// mobject-datatypes/Primitive/_LWORD
{attribute 'linkalways'} 
{attribute 'no_explicit_call' := 'This FB is a CLASS and must be accessed using methods or properties'}
{attribute 'enable_dynamic_creation'}
FUNCTION_BLOCK _LWORD EXTENDS NumericDatatypeBase
VAR
	localData : LWORD;
	activeData : REFERENCE TO LWORD REF= localData;
END_VAR

METHOD FB_init : BOOL
VAR_INPUT
	bInitRetains : BOOL; // if TRUE, the retain variables are initialized (warm start / cold start)
	bInCopyCode : BOOL;  // if TRUE, the instance afterwards gets moved WORDo the copy code (online change)
	InitialValue : LWORD;
END_VAR
localData := InitialValue;
END_METHOD

METHOD PROTECTED SerializeMaxValue
VAR_INPUT
	Serializer : I_Serializer;
END_VAR
Serializer.AddLword(MaxValue);
END_METHOD

METHOD PROTECTED SerializeMinValue
VAR_INPUT
	Serializer : I_Serializer;
END_VAR
Serializer.AddLword(MinValue);
END_METHOD

PROPERTY PUBLIC Address : PVOID
GET
Address := ADR(activeData);
END_GET
END_PROPERTY

METHOD PUBLIC ClearReference
VAR_INPUT
END_VAR
activeData REF= localData;
END_METHOD

METHOD PUBLIC Clone : I_Datatype
VAR
    pClone : POINTER TO _LWORD;
END_VAR
pClone := __NEW(_LWORD(InitialValue := Value));
Clone := pClone^;
END_METHOD

PROPERTY PUBLIC IsEven : BOOL
GET
IsEven := (Value mod 2) = 0;
END_GET
END_PROPERTY

PROPERTY PUBLIC IsFloat : BOOL
GET
IsFloat := FALSE;
END_GET
END_PROPERTY

PROPERTY PUBLIC IsSigned : BOOL
GET
IsSigned := FALSE;
END_GET
END_PROPERTY

METHOD PUBLIC MakeReferenceTo
VAR_INPUT
	ReferenceTarget : REFERENCE TO LWORD;
END_VAR
activeData REF= ReferenceTarget;
END_METHOD

PROPERTY PUBLIC MaxValue : LWORD
GET
MaxValue :=  DatatypeLimits.LWORD_MAX_VALUE;
END_GET
END_PROPERTY

PROPERTY PUBLIC MinValue : LWORD
GET
MinValue := DatatypeLimits.LWORD_MIN_VALUE;
END_GET
END_PROPERTY

METHOD PUBLIC SerializeWith
VAR_INPUT
	Serializer : I_Serializer;
END_VAR
Serializer.AddLword(activeData);
END_METHOD

PROPERTY PUBLIC Size : UDINT
GET
Size := SIZEOF(activeData);
END_GET
END_PROPERTY

METHOD TryDeserializeFrom : BOOL
VAR_INPUT
	Deserializer : I_Deserializer;
	Feedback : I_DeserializerFeedback;
END_VAR
TryDeserializeFrom := Deserializer.TryGetLword(activeData, Feedback);
END_METHOD

METHOD TryMakeReferenceTo : BOOL
VAR_INPUT
	Target : I_Datatype;
END_VAR
VAR
	pTargetData : POINTER TO LWORD;
END_VAR
IF NOT IsEquivalentTo(Target) THEN
	RETURN;
END_IF

pTargetData := Target.Address;
activeData REF= pTargetData^;
TryMakeReferenceTo := TRUE;
END_METHOD

PROPERTY PUBLIC TypeName : T_MAXSTRING
GET
TypeName := 'LWORD';
END_GET
END_PROPERTY

PROPERTY PUBLIC Value : REFERENCE TO LWORD
GET
Value REF= activeData;
END_GET
END_PROPERTY

END_FUNCTION_BLOCK

// mobject-converters/Converters/BOOL_TO_/TryConvert_BOOL_TO_SINT
FUNCTION TryConvert_BOOL_TO_SINT : BOOL
VAR_INPUT
	in : BOOL;
	out : REFERENCE TO SINT;
END_VAR

out := BOOL_TO_SINT(in);
TryConvert_BOOL_TO_SINT := TRUE;

END_FUNCTION

// mobject-datatypes/Primitive/_SINT
{attribute 'linkalways'} 
{attribute 'no_explicit_call' := 'This FB is a CLASS and must be accessed using methods or properties'}
{attribute 'enable_dynamic_creation'}
FUNCTION_BLOCK _SINT EXTENDS NumericDatatypeBase
VAR
	localData : SINT;
	activeData : REFERENCE TO SINT REF= localData;
END_VAR

METHOD FB_init : BOOL
VAR_INPUT
	bInitRetains : BOOL; // if TRUE, the retain variables are initialized (warm start / cold start)
	bInCopyCode : BOOL;  // if TRUE, the instance afterwards gets moved into the copy code (online change)
	InitialValue : SINT;
END_VAR
localData := InitialValue;
END_METHOD

METHOD PROTECTED SerializeMaxValue
VAR_INPUT
	Serializer : I_Serializer;
END_VAR
Serializer.AddSint(MaxValue);
END_METHOD

METHOD PROTECTED SerializeMinValue
VAR_INPUT
	Serializer : I_Serializer;
END_VAR
Serializer.AddSint(MinValue);
END_METHOD

PROPERTY PUBLIC Address : PVOID
GET
Address := ADR(activeData);
END_GET
END_PROPERTY

METHOD PUBLIC ClearReference
VAR_INPUT
END_VAR
activeData REF= localData;
END_METHOD

METHOD PUBLIC Clone : I_Datatype
VAR
    pClone : POINTER TO _SINT;
END_VAR
pClone := __NEW(_SINT(InitialValue := Value));
Clone := pClone^;
END_METHOD

PROPERTY PUBLIC IsEven : BOOL
GET
IsEven := (Value mod 2) = 0;
END_GET
END_PROPERTY

PROPERTY PUBLIC IsFloat : BOOL
GET
IsFloat := FALSE;
END_GET
END_PROPERTY

PROPERTY PUBLIC IsSigned : BOOL
GET
IsSigned := TRUE;
END_GET
END_PROPERTY

METHOD PUBLIC MakeReferenceTo
VAR_INPUT
	ReferenceTarget : REFERENCE TO SINT;
END_VAR
activeData REF= ReferenceTarget;
END_METHOD

PROPERTY PUBLIC MaxValue : SINT
GET
MaxValue :=  DatatypeLimits.SINT_MAX_VALUE;
END_GET
END_PROPERTY

PROPERTY PUBLIC MinValue : SINT
GET
MinValue := DatatypeLimits.SINT_MIN_VALUE;
END_GET
END_PROPERTY

METHOD PUBLIC SerializeWith
VAR_INPUT
	Serializer : I_Serializer;
END_VAR
Serializer.AddSint(activeData);
END_METHOD

PROPERTY PUBLIC Size : UDINT
GET
Size := SIZEOF(activeData);
END_GET
END_PROPERTY

METHOD TryDeserializeFrom : BOOL
VAR_INPUT
	Deserializer : I_Deserializer;
	Feedback : I_DeserializerFeedback;
END_VAR
TryDeserializeFrom := Deserializer.TryGetSint(activeData, Feedback);
END_METHOD

METHOD TryMakeReferenceTo : BOOL
VAR_INPUT
	Target : I_Datatype;
END_VAR
VAR
	pTargetData : POINTER TO SINT;
END_VAR
IF NOT IsEquivalentTo(Target) THEN
	RETURN;
END_IF

pTargetData := Target.Address;
activeData REF= pTargetData^;
TryMakeReferenceTo := TRUE;
END_METHOD

PROPERTY PUBLIC TypeName : T_MAXSTRING
GET
TypeName := 'SINT';
END_GET
END_PROPERTY

PROPERTY PUBLIC Value : REFERENCE TO SINT
GET
Value REF= activeData;
END_GET
END_PROPERTY

END_FUNCTION_BLOCK

// mobject-converters/Converters/BOOL_TO_/TryConvert_BOOL_TO_INT
FUNCTION TryConvert_BOOL_TO_INT : BOOL
VAR_INPUT
	in : BOOL;
	out : REFERENCE TO INT;
END_VAR

out := BOOL_TO_INT(in);
TryConvert_BOOL_TO_INT := TRUE;

END_FUNCTION

// mobject-datatypes/Primitive/_INT
{attribute 'linkalways'} 
{attribute 'no_explicit_call' := 'This FB is a CLASS and must be accessed using methods or properties'}
{attribute 'enable_dynamic_creation'}
FUNCTION_BLOCK _INT EXTENDS NumericDatatypeBase
VAR
	localData : INT;
	activeData : REFERENCE TO INT REF= localData;
END_VAR

METHOD FB_init : BOOL
VAR_INPUT
	bInitRetains : BOOL; // if TRUE, the retain variables are initialized (warm start / cold start)
	bInCopyCode : BOOL;  // if TRUE, the instance afterwards gets moved into the copy code (online change)
	InitialValue : INT;
END_VAR
localData := InitialValue;
END_METHOD

METHOD PROTECTED SerializeMaxValue
VAR_INPUT
	Serializer : I_Serializer;
END_VAR
Serializer.AddInt(MaxValue);
END_METHOD

METHOD PROTECTED SerializeMinValue
VAR_INPUT
	Serializer : I_Serializer;
END_VAR
Serializer.AddInt(MinValue);
END_METHOD

PROPERTY PUBLIC Address : PVOID
GET
Address := ADR(activeData);
END_GET
END_PROPERTY

METHOD PUBLIC ClearReference
VAR_INPUT
END_VAR
activeData REF= localData;
END_METHOD

METHOD PUBLIC Clone : I_Datatype
VAR
    pClone : POINTER TO _INT;
END_VAR
pClone := __NEW(_INT(InitialValue := Value));
Clone := pClone^;
END_METHOD

PROPERTY PUBLIC IsEven : BOOL
GET
IsEven := (Value mod 2) = 0;
END_GET
END_PROPERTY

PROPERTY PUBLIC IsFloat : BOOL
GET
IsFloat := FALSE;
END_GET
END_PROPERTY

PROPERTY PUBLIC IsSigned : BOOL
GET
IsSigned := TRUE;
END_GET
END_PROPERTY

METHOD PUBLIC MakeReferenceTo
VAR_INPUT
	ReferenceTarget : REFERENCE TO INT;
END_VAR
activeData REF= ReferenceTarget;
END_METHOD

PROPERTY PUBLIC MaxValue : INT
GET
MaxValue := DatatypeLimits.INT_MAX_VALUE;
END_GET
END_PROPERTY

PROPERTY PUBLIC MinValue : INT
GET
MinValue := DatatypeLimits.INT_MIN_VALUE;
END_GET
END_PROPERTY

METHOD PUBLIC SerializeWith
VAR_INPUT
	Serializer : I_Serializer;
END_VAR
Serializer.AddInt(activeData);
END_METHOD

PROPERTY PUBLIC Size : UDINT
GET
Size := SIZEOF(activeData);
END_GET
END_PROPERTY

METHOD TryDeserializeFrom : BOOL
VAR_INPUT
	Deserializer : I_Deserializer;
	Feedback : I_DeserializerFeedback;
END_VAR
TryDeserializeFrom := Deserializer.TryGetInt(activeData, Feedback);
END_METHOD

METHOD TryMakeReferenceTo : BOOL
VAR_INPUT
	Target : I_Datatype;
END_VAR
VAR
	pTargetData : POINTER TO INT;
END_VAR
IF NOT IsEquivalentTo(Target) THEN
	RETURN;
END_IF

pTargetData := Target.Address;
activeData REF= pTargetData^;
TryMakeReferenceTo := TRUE;
END_METHOD

PROPERTY PUBLIC TypeName : T_MAXSTRING
GET
TypeName := 'INT';
END_GET
END_PROPERTY

PROPERTY PUBLIC Value : REFERENCE TO INT
GET
Value REF= activeData;
END_GET
END_PROPERTY

END_FUNCTION_BLOCK

// mobject-converters/Converters/BOOL_TO_/TryConvert_BOOL_TO_DINT
FUNCTION TryConvert_BOOL_TO_DINT : BOOL
VAR_INPUT
	in : BOOL;
	out : REFERENCE TO DINT;
END_VAR

out := BOOL_TO_DINT(in);
TryConvert_BOOL_TO_DINT := TRUE;

END_FUNCTION

// mobject-datatypes/Primitive/_DINT
{attribute 'linkalways'} 
{attribute 'no_explicit_call' := 'This FB is a CLASS and must be accessed using methods or properties'}
{attribute 'enable_dynamic_creation'}
FUNCTION_BLOCK _DINT EXTENDS NumericDatatypeBase
VAR
	localData : DINT;
	activeData : REFERENCE TO DINT REF= localData;
END_VAR

METHOD FB_init : BOOL
VAR_INPUT
	bInitRetains : BOOL; // if TRUE, the retain variables are initialized (warm start / cold start)
	bInCopyCode : BOOL;  // if TRUE, the instance afterwards gets moved into the copy code (online change)
	InitialValue : DINT;
END_VAR
localData := InitialValue;
END_METHOD

METHOD PROTECTED SerializeMaxValue
VAR_INPUT
	Serializer : I_Serializer;
END_VAR
Serializer.AddDint(MaxValue);
END_METHOD

METHOD PROTECTED SerializeMinValue
VAR_INPUT
	Serializer : I_Serializer;
END_VAR
Serializer.AddDint(MinValue);
END_METHOD

PROPERTY PUBLIC Address : PVOID
GET
Address := ADR(activeData);
END_GET
END_PROPERTY

METHOD PUBLIC ClearReference
VAR_INPUT
END_VAR
activeData REF= localData;
END_METHOD

METHOD PUBLIC Clone : I_Datatype
VAR
    pClone : POINTER TO _DINT;
END_VAR
pClone := __NEW(_DINT(InitialValue := Value));
Clone := pClone^;
END_METHOD

PROPERTY PUBLIC IsEven : BOOL
GET
IsEven := (Value mod 2) = 0;
END_GET
END_PROPERTY

PROPERTY PUBLIC IsFloat : BOOL
GET
IsFloat := FALSE;
END_GET
END_PROPERTY

PROPERTY PUBLIC IsSigned : BOOL
GET
IsSigned := TRUE;
END_GET
END_PROPERTY

METHOD PUBLIC MakeReferenceTo
VAR_INPUT
	ReferenceTarget : REFERENCE TO DINT;
END_VAR
activeData REF= ReferenceTarget;
END_METHOD

PROPERTY PUBLIC MaxValue : DINT
GET
MaxValue := DatatypeLimits.DINT_MAX_VALUE;
END_GET
END_PROPERTY

PROPERTY PUBLIC MinValue : DINT
GET
MinValue := DatatypeLimits.DINT_MIN_VALUE;
END_GET
END_PROPERTY

METHOD PUBLIC SerializeWith
VAR_INPUT
	Serializer : I_Serializer;
END_VAR
Serializer.AddDint(activeData);
END_METHOD

PROPERTY PUBLIC Size : UDINT
GET
Size := SIZEOF(activeData);
END_GET
END_PROPERTY

METHOD TryDeserializeFrom : BOOL
VAR_INPUT
	Deserializer : I_Deserializer;
	Feedback : I_DeserializerFeedback;
END_VAR
TryDeserializeFrom := Deserializer.TryGetDint(activeData, Feedback);
END_METHOD

METHOD TryMakeReferenceTo : BOOL
VAR_INPUT
	Target : I_Datatype;
END_VAR
VAR
	pTargetData : POINTER TO DINT;
END_VAR
IF NOT IsEquivalentTo(Target) THEN
	RETURN;
END_IF

pTargetData := Target.Address;
activeData REF= pTargetData^;
TryMakeReferenceTo := TRUE;
END_METHOD

PROPERTY PUBLIC TypeName : T_MAXSTRING
GET
TypeName := 'DINT';
END_GET
END_PROPERTY

PROPERTY PUBLIC Value : REFERENCE TO DINT
GET
Value REF= activeData;
END_GET
END_PROPERTY

END_FUNCTION_BLOCK

// mobject-converters/Converters/BOOL_TO_/TryConvert_BOOL_TO_LINT
FUNCTION TryConvert_BOOL_TO_LINT : BOOL
VAR_INPUT
	in : BOOL;
	out : REFERENCE TO LINT;
END_VAR

out := BOOL_TO_LINT(in);
TryConvert_BOOL_TO_LINT := TRUE;

END_FUNCTION

// mobject-datatypes/Primitive/_LINT
{attribute 'linkalways'} 
{attribute 'no_explicit_call' := 'This FB is a CLASS and must be accessed using methods or properties'}
{attribute 'enable_dynamic_creation'}
FUNCTION_BLOCK _LINT EXTENDS NumericDatatypeBase
VAR
	localData : LINT;
	activeData : REFERENCE TO LINT REF= localData;
END_VAR

METHOD FB_init : BOOL
VAR_INPUT
	bInitRetains : BOOL; // if TRUE, the retain variables are initialized (warm start / cold start)
	bInCopyCode : BOOL;  // if TRUE, the instance afterwards gets moved into the copy code (online change)
	InitialValue : LINT;
END_VAR
localData := InitialValue;
END_METHOD

METHOD PROTECTED SerializeMaxValue
VAR_INPUT
	Serializer : I_Serializer;
END_VAR
Serializer.AddLint(MaxValue);
END_METHOD

METHOD PROTECTED SerializeMinValue
VAR_INPUT
	Serializer : I_Serializer;
END_VAR
Serializer.AddLint(MinValue);
END_METHOD

PROPERTY PUBLIC Address : PVOID
GET
Address := ADR(activeData);
END_GET
END_PROPERTY

METHOD PUBLIC ClearReference
VAR_INPUT
END_VAR
activeData REF= localData;
END_METHOD

METHOD PUBLIC Clone : I_Datatype
VAR
    pClone : POINTER TO _LINT;
END_VAR
pClone := __NEW(_LINT(InitialValue := Value));
Clone := pClone^;
END_METHOD

PROPERTY PUBLIC IsEven : BOOL
GET
IsEven := (Value mod 2) = 0;
END_GET
END_PROPERTY

PROPERTY PUBLIC IsFloat : BOOL
GET
IsFloat := FALSE;
END_GET
END_PROPERTY

PROPERTY PUBLIC IsSigned : BOOL
GET
IsSigned := TRUE;
END_GET
END_PROPERTY

METHOD PUBLIC MakeReferenceTo
VAR_INPUT
	ReferenceTarget : REFERENCE TO LINT;
END_VAR
activeData REF= ReferenceTarget;
END_METHOD

PROPERTY PUBLIC MaxValue : LINT
GET
MaxValue :=  DatatypeLimits.LINT_MAX_VALUE;
END_GET
END_PROPERTY

PROPERTY PUBLIC MinValue : LINT
GET
MinValue := DatatypeLimits.LINT_MIN_VALUE;
END_GET
END_PROPERTY

METHOD PUBLIC SerializeWith
VAR_INPUT
	Serializer : I_Serializer;
END_VAR
Serializer.AddLint(activeData);
END_METHOD

PROPERTY PUBLIC Size : UDINT
GET
Size := SIZEOF(activeData);
END_GET
END_PROPERTY

METHOD TryDeserializeFrom : BOOL
VAR_INPUT
	Deserializer : I_Deserializer;
	Feedback : I_DeserializerFeedback;
END_VAR
TryDeserializeFrom := Deserializer.TryGetLint(activeData, Feedback);
END_METHOD

METHOD TryMakeReferenceTo : BOOL
VAR_INPUT
	Target : I_Datatype;
END_VAR
VAR
	pTargetData : POINTER TO LINT;
END_VAR
IF NOT IsEquivalentTo(Target) THEN
	RETURN;
END_IF

pTargetData := Target.Address;
activeData REF= pTargetData^;
TryMakeReferenceTo := TRUE;
END_METHOD

PROPERTY PUBLIC TypeName : T_MAXSTRING
GET
TypeName := 'LINT';
END_GET
END_PROPERTY

PROPERTY PUBLIC Value : REFERENCE TO LINT
GET
Value REF= activeData;
END_GET
END_PROPERTY

END_FUNCTION_BLOCK

// mobject-converters/Converters/BOOL_TO_/TryConvert_BOOL_TO_USINT
FUNCTION TryConvert_BOOL_TO_USINT : BOOL
VAR_INPUT
	in : BOOL;
	out : REFERENCE TO USINT;
END_VAR

out := BOOL_TO_USINT(in);
TryConvert_BOOL_TO_USINT := TRUE;

END_FUNCTION

// mobject-datatypes/Primitive/_USINT
{attribute 'linkalways'} 
{attribute 'no_explicit_call' := 'This FB is a CLASS and must be accessed using methods or properties'}
{attribute 'enable_dynamic_creation'}
FUNCTION_BLOCK _USINT EXTENDS NumericDatatypeBase
VAR
	localData : USINT;
	activeData : REFERENCE TO USINT REF= localData;
END_VAR

METHOD FB_init : BOOL
VAR_INPUT
	bInitRetains : BOOL; // if TRUE, the retain variables are initialized (warm start / cold start)
	bInCopyCode : BOOL;  // if TRUE, the instance afterwards gets moved into the copy code (online change)
	InitialValue : USINT;
END_VAR
localData := InitialValue;
END_METHOD

METHOD PROTECTED SerializeMaxValue
VAR_INPUT
	Serializer : I_Serializer;
END_VAR
Serializer.AddUsint(MaxValue);
END_METHOD

METHOD PROTECTED SerializeMinValue
VAR_INPUT
	Serializer : I_Serializer;
END_VAR
Serializer.AddUsint(MinValue);
END_METHOD

PROPERTY PUBLIC Address : PVOID
GET
Address := ADR(activeData);
END_GET
END_PROPERTY

METHOD PUBLIC ClearReference
VAR_INPUT
END_VAR
activeData REF= localData;
END_METHOD

METHOD PUBLIC Clone : I_Datatype
VAR
    pClone : POINTER TO _USINT;
END_VAR
pClone := __NEW(_USINT(InitialValue := Value));
Clone := pClone^;
END_METHOD

PROPERTY PUBLIC IsEven : BOOL
GET
IsEven := (Value mod 2) = 0;
END_GET
END_PROPERTY

PROPERTY PUBLIC IsFloat : BOOL
GET
IsFloat := FALSE;
END_GET
END_PROPERTY

PROPERTY PUBLIC IsSigned : BOOL
GET
IsSigned := FALSE;
END_GET
END_PROPERTY

METHOD PUBLIC MakeReferenceTo
VAR_INPUT
	ReferenceTarget : REFERENCE TO USINT;
END_VAR
activeData REF= ReferenceTarget;
END_METHOD

PROPERTY PUBLIC MaxValue : USINT
GET
MaxValue :=  DatatypeLimits.USINT_MAX_VALUE;
END_GET
END_PROPERTY

PROPERTY PUBLIC MinValue : USINT
GET
MinValue := DatatypeLimits.USINT_MIN_VALUE;
END_GET
END_PROPERTY

METHOD PUBLIC SerializeWith
VAR_INPUT
	Serializer : I_Serializer;
END_VAR
Serializer.AddUsint(activeData);
END_METHOD

PROPERTY PUBLIC Size : UDINT
GET
Size := SIZEOF(activeData);
END_GET
END_PROPERTY

METHOD TryDeserializeFrom : BOOL
VAR_INPUT
	Deserializer : I_Deserializer;
	Feedback : I_DeserializerFeedback;
END_VAR
TryDeserializeFrom := Deserializer.TryGetUsint(activeData, Feedback);
END_METHOD

METHOD TryMakeReferenceTo : BOOL
VAR_INPUT
	Target : I_Datatype;
END_VAR
VAR
	pTargetData : POINTER TO USINT;
END_VAR
IF NOT IsEquivalentTo(Target) THEN
	RETURN;
END_IF

pTargetData := Target.Address;
activeData REF= pTargetData^;
TryMakeReferenceTo := TRUE;
END_METHOD

PROPERTY PUBLIC TypeName : T_MAXSTRING
GET
TypeName := 'USINT';
END_GET
END_PROPERTY

PROPERTY PUBLIC Value : REFERENCE TO USINT
GET
Value REF= activeData;
END_GET
END_PROPERTY

END_FUNCTION_BLOCK

// mobject-converters/Converters/BOOL_TO_/TryConvert_BOOL_TO_UINT
FUNCTION TryConvert_BOOL_TO_UINT : BOOL
VAR_INPUT
	in : BOOL;
	out : REFERENCE TO UINT;
END_VAR

out := BOOL_TO_UINT(in);
TryConvert_BOOL_TO_UINT := TRUE;

END_FUNCTION

// mobject-datatypes/Primitive/_UINT
{attribute 'linkalways'} 
{attribute 'no_explicit_call' := 'This FB is a CLASS and must be accessed using methods or properties'}
{attribute 'enable_dynamic_creation'}
FUNCTION_BLOCK _UINT EXTENDS NumericDatatypeBase
VAR
	localData : UINT;
	activeData : REFERENCE TO UINT REF= localData;
END_VAR

METHOD FB_init : BOOL
VAR_INPUT
	bInitRetains : BOOL; // if TRUE, the retain variables are initialized (warm start / cold start)
	bInCopyCode : BOOL;  // if TRUE, the instance afterwards gets moved into the copy code (online change)
	InitialValue : UINT;
END_VAR
localData := InitialValue;
END_METHOD

METHOD PROTECTED SerializeMaxValue
VAR_INPUT
	Serializer : I_Serializer;
END_VAR
Serializer.AddUint(MaxValue);
END_METHOD

METHOD PROTECTED SerializeMinValue
VAR_INPUT
	Serializer : I_Serializer;
END_VAR
Serializer.AddUint(MinValue);
END_METHOD

PROPERTY PUBLIC Address : PVOID
GET
Address := ADR(activeData);
END_GET
END_PROPERTY

METHOD PUBLIC ClearReference
VAR_INPUT
END_VAR
activeData REF= localData;
END_METHOD

METHOD PUBLIC Clone : I_Datatype
VAR
    pClone : POINTER TO _UINT;
END_VAR
pClone := __NEW(_UINT(InitialValue := Value));
Clone := pClone^;
END_METHOD

PROPERTY PUBLIC IsEven : BOOL
GET
IsEven := (Value mod 2) = 0;
END_GET
END_PROPERTY

PROPERTY PUBLIC IsFloat : BOOL
GET
IsFloat := FALSE;
END_GET
END_PROPERTY

PROPERTY PUBLIC IsSigned : BOOL
GET
IsSigned := FALSE;
END_GET
END_PROPERTY

METHOD PUBLIC MakeReferenceTo
VAR_INPUT
	ReferenceTarget : REFERENCE TO UINT;
END_VAR
activeData REF= ReferenceTarget;
END_METHOD

PROPERTY PUBLIC MaxValue : UINT
GET
MaxValue :=  DatatypeLimits.UINT_MAX_VALUE;
END_GET
END_PROPERTY

PROPERTY PUBLIC MinValue : UINT
GET
MinValue := DatatypeLimits.UINT_MIN_VALUE;
END_GET
END_PROPERTY

METHOD PUBLIC SerializeWith
VAR_INPUT
	Serializer : I_Serializer;
END_VAR
Serializer.AddUint(activeData);
END_METHOD

PROPERTY PUBLIC Size : UDINT
GET
Size := SIZEOF(activeData);
END_GET
END_PROPERTY

METHOD TryDeserializeFrom : BOOL
VAR_INPUT
	Deserializer : I_Deserializer;
	Feedback : I_DeserializerFeedback;
END_VAR
TryDeserializeFrom := Deserializer.TryGetUint(activeData, Feedback);
END_METHOD

METHOD TryMakeReferenceTo : BOOL
VAR_INPUT
	Target : I_Datatype;
END_VAR
VAR
	pTargetData : POINTER TO UINT;
END_VAR
IF NOT IsEquivalentTo(Target) THEN
	RETURN;
END_IF

pTargetData := Target.Address;
activeData REF= pTargetData^;
TryMakeReferenceTo := TRUE;
END_METHOD

PROPERTY PUBLIC TypeName : T_MAXSTRING
GET
TypeName := 'UINT';
END_GET
END_PROPERTY

PROPERTY PUBLIC Value : REFERENCE TO UINT
GET
Value REF= activeData;
END_GET
END_PROPERTY

END_FUNCTION_BLOCK

// mobject-converters/Converters/BOOL_TO_/TryConvert_BOOL_TO_UDINT
FUNCTION TryConvert_BOOL_TO_UDINT : BOOL
VAR_INPUT
	in : BOOL;
	out : REFERENCE TO UDINT;
END_VAR

out := BOOL_TO_UDINT(in);
TryConvert_BOOL_TO_UDINT := TRUE;

END_FUNCTION

// mobject-datatypes/Primitive/_UDINT
{attribute 'linkalways'} 
{attribute 'no_explicit_call' := 'This FB is a CLASS and must be accessed using methods or properties'}
{attribute 'enable_dynamic_creation'}
FUNCTION_BLOCK _UDINT EXTENDS NumericDatatypeBase
VAR
	localData : UDINT;
	activeData : REFERENCE TO UDINT REF= localData;
END_VAR

METHOD FB_init : BOOL
VAR_INPUT
	bInitRetains : BOOL; // if TRUE, the retain variables are initialized (warm start / cold start)
	bInCopyCode : BOOL;  // if TRUE, the instance afterwards gets moved into the copy code (online change)
	InitialValue : UDINT;
END_VAR
localData := InitialValue;
END_METHOD

METHOD PROTECTED SerializeMaxValue
VAR_INPUT
	Serializer : I_Serializer;
END_VAR
Serializer.AddUdint(MaxValue);
END_METHOD

METHOD PROTECTED SerializeMinValue
VAR_INPUT
	Serializer : I_Serializer;
END_VAR
Serializer.AddUdint(MinValue);
END_METHOD

PROPERTY PUBLIC Address : PVOID
GET
Address := ADR(activeData);
END_GET
END_PROPERTY

METHOD PUBLIC ClearReference
VAR_INPUT
END_VAR
activeData REF= localData;
END_METHOD

METHOD PUBLIC Clone : I_Datatype
VAR
    pClone : POINTER TO _UDINT;
END_VAR
pClone := __NEW(_UDINT(InitialValue := Value));
Clone := pClone^;
END_METHOD

PROPERTY PUBLIC IsEven : BOOL
GET
IsEven := (Value mod 2) = 0;
END_GET
END_PROPERTY

PROPERTY PUBLIC IsFloat : BOOL
GET
IsFloat := FALSE;
END_GET
END_PROPERTY

PROPERTY PUBLIC IsSigned : BOOL
GET
IsSigned := FALSE;
END_GET
END_PROPERTY

METHOD PUBLIC MakeReferenceTo
VAR_INPUT
	ReferenceTarget : REFERENCE TO UDINT;
END_VAR
activeData REF= ReferenceTarget;
END_METHOD

PROPERTY PUBLIC MaxValue : UDINT
GET
MaxValue :=  DatatypeLimits.UDINT_MAX_VALUE;
END_GET
END_PROPERTY

PROPERTY PUBLIC MinValue : UDINT
GET
MinValue := DatatypeLimits.UDINT_MIN_VALUE;
END_GET
END_PROPERTY

METHOD PUBLIC SerializeWith
VAR_INPUT
	Serializer : I_Serializer;
END_VAR
Serializer.AddUdint(activeData);
END_METHOD

PROPERTY PUBLIC Size : UDINT
GET
Size := SIZEOF(activeData);
END_GET
END_PROPERTY

METHOD TryDeserializeFrom : BOOL
VAR_INPUT
	Deserializer : I_Deserializer;
	Feedback : I_DeserializerFeedback;
END_VAR
TryDeserializeFrom := Deserializer.TryGetUdint(activeData, Feedback);
END_METHOD

METHOD TryMakeReferenceTo : BOOL
VAR_INPUT
	Target : I_Datatype;
END_VAR
VAR
	pTargetData : POINTER TO UDINT;
END_VAR
IF NOT IsEquivalentTo(Target) THEN
	RETURN;
END_IF

pTargetData := Target.Address;
activeData REF= pTargetData^;
TryMakeReferenceTo := TRUE;
END_METHOD

PROPERTY PUBLIC TypeName : T_MAXSTRING
GET
TypeName := 'UDINT';
END_GET
END_PROPERTY

PROPERTY PUBLIC Value : REFERENCE TO UDINT
GET
Value REF= activeData;
END_GET
END_PROPERTY

END_FUNCTION_BLOCK

// mobject-converters/Converters/BOOL_TO_/TryConvert_BOOL_TO_ULINT
FUNCTION TryConvert_BOOL_TO_ULINT : BOOL
VAR_INPUT
	in : BOOL;
	out : REFERENCE TO ULINT;
END_VAR

out := BOOL_TO_ULINT(in);
TryConvert_BOOL_TO_ULINT := TRUE;

END_FUNCTION

// mobject-datatypes/Primitive/_ULINT
{attribute 'linkalways'} 
{attribute 'no_explicit_call' := 'This FB is a CLASS and must be accessed using methods or properties'}
{attribute 'enable_dynamic_creation'}
FUNCTION_BLOCK _ULINT EXTENDS NumericDatatypeBase
VAR
	localData : ULINT;
	activeData : REFERENCE TO ULINT REF= localData;
END_VAR

METHOD FB_init : BOOL
VAR_INPUT
	bInitRetains : BOOL; // if TRUE, the retain variables are initialized (warm start / cold start)
	bInCopyCode : BOOL;  // if TRUE, the instance afterwards gets moved into the copy code (online change)
	InitialValue : ULINT;
END_VAR
localData := InitialValue;
END_METHOD

METHOD PROTECTED SerializeMaxValue
VAR_INPUT
	Serializer : I_Serializer;
END_VAR
Serializer.AddUlint(MaxValue);
END_METHOD

METHOD PROTECTED SerializeMinValue
VAR_INPUT
	Serializer : I_Serializer;
END_VAR
Serializer.AddUlint(MinValue);
END_METHOD

PROPERTY PUBLIC Address : PVOID
GET
Address := ADR(activeData);
END_GET
END_PROPERTY

METHOD PUBLIC ClearReference
VAR_INPUT
END_VAR
activeData REF= localData;
END_METHOD

METHOD PUBLIC Clone : I_Datatype
VAR
    pClone : POINTER TO _ULINT;
END_VAR
pClone := __NEW(_ULINT(InitialValue := Value));
Clone := pClone^;
END_METHOD

PROPERTY PUBLIC IsEven : BOOL
GET
IsEven := (Value mod 2) = 0;
END_GET
END_PROPERTY

PROPERTY PUBLIC IsFloat : BOOL
GET
IsFloat := FALSE;
END_GET
END_PROPERTY

PROPERTY PUBLIC IsSigned : BOOL
GET
IsSigned := FALSE;
END_GET
END_PROPERTY

METHOD PUBLIC MakeReferenceTo
VAR_INPUT
	ReferenceTarget : REFERENCE TO ULINT;
END_VAR
activeData REF= ReferenceTarget;
END_METHOD

PROPERTY PUBLIC MaxValue : ULINT
GET
MaxValue :=  DatatypeLimits.ULINT_MAX_VALUE;
END_GET
END_PROPERTY

PROPERTY PUBLIC MinValue : ULINT
GET
MinValue := DatatypeLimits.ULINT_MIN_VALUE;
END_GET
END_PROPERTY

METHOD PUBLIC SerializeWith
VAR_INPUT
	Serializer : I_Serializer;
END_VAR
Serializer.AddUlint(activeData);
END_METHOD

PROPERTY PUBLIC Size : UDINT
GET
Size := SIZEOF(activeData);
END_GET
END_PROPERTY

METHOD TryDeserializeFrom : BOOL
VAR_INPUT
	Deserializer : I_Deserializer;
	Feedback : I_DeserializerFeedback;
END_VAR
TryDeserializeFrom := Deserializer.TryGetUlint(activeData, Feedback);
END_METHOD

METHOD TryMakeReferenceTo : BOOL
VAR_INPUT
	Target : I_Datatype;
END_VAR
VAR
	pTargetData : POINTER TO ULINT;
END_VAR
IF NOT IsEquivalentTo(Target) THEN
	RETURN;
END_IF

pTargetData := Target.Address;
activeData REF= pTargetData^;
TryMakeReferenceTo := TRUE;
END_METHOD

PROPERTY PUBLIC TypeName : T_MAXSTRING
GET
TypeName := 'ULINT';
END_GET
END_PROPERTY

PROPERTY PUBLIC Value : REFERENCE TO ULINT
GET
Value REF= activeData;
END_GET
END_PROPERTY

END_FUNCTION_BLOCK

// mobject-converters/Converters/BOOL_TO_/TryConvert_BOOL_TO_REAL
FUNCTION TryConvert_BOOL_TO_REAL : BOOL
VAR_INPUT
	in : BOOL;
	out : REFERENCE TO REAL;
END_VAR

out := BOOL_TO_REAL(in);
TryConvert_BOOL_TO_REAL := TRUE;

END_FUNCTION

// mobject-datatypes/Primitive/_REAL
{attribute 'linkalways'} 
{attribute 'no_explicit_call' := 'This FB is a CLASS and must be accessed using methods or properties'}
{attribute 'enable_dynamic_creation'}
FUNCTION_BLOCK _REAL EXTENDS NumericDatatypeBase
VAR
	localData : REAL;
	activeData : REFERENCE TO REAL REF= localData;
END_VAR

METHOD FB_init : BOOL
VAR_INPUT
	bInitRetains : BOOL; // if TRUE, the retain variables are initialized (warm start / cold start)
	bInCopyCode : BOOL;  // if TRUE, the instance afterwards gets moved into the copy code (online change)
	InitialValue : REAL;
END_VAR
localData := InitialValue;
END_METHOD

METHOD PROTECTED SerializeMaxValue
VAR_INPUT
	Serializer : I_Serializer;
END_VAR
Serializer.AddReal(MaxValue);
END_METHOD

METHOD PROTECTED SerializeMinValue
VAR_INPUT
	Serializer : I_Serializer;
END_VAR
Serializer.AddReal(MinValue);
END_METHOD

PROPERTY PUBLIC Address : PVOID
GET
Address := ADR(activeData);
END_GET
END_PROPERTY

METHOD PUBLIC ClearReference
VAR_INPUT
END_VAR
activeData REF= localData;
END_METHOD

METHOD PUBLIC Clone : I_Datatype
VAR
    pClone : POINTER TO _REAL;
END_VAR
pClone := __NEW(_REAL(InitialValue := Value));
Clone := pClone^;
END_METHOD

PROPERTY PUBLIC IsEven : BOOL
GET
IsEven := FALSE;
END_GET
END_PROPERTY

PROPERTY PUBLIC IsFloat : BOOL
GET
IsFloat := TRUE;
END_GET
END_PROPERTY

PROPERTY PUBLIC IsOdd : BOOL
GET
IsOdd := FALSE;
END_GET
END_PROPERTY

PROPERTY PUBLIC IsSigned : BOOL
GET
IsSigned := TRUE;
END_GET
END_PROPERTY

METHOD PUBLIC MakeReferenceTo
VAR_INPUT
	ReferenceTarget : REFERENCE TO REAL;
END_VAR
activeData REF= ReferenceTarget;
END_METHOD

PROPERTY PUBLIC MaxValue : REAL
GET
MaxValue :=  DatatypeLimits.REAL_MAX_VALUE;
END_GET
END_PROPERTY

PROPERTY PUBLIC MinValue : REAL
GET
MinValue := DatatypeLimits.REAL_MIN_VALUE;
END_GET
END_PROPERTY

METHOD PUBLIC SerializeWith
VAR_INPUT
	Serializer : I_Serializer;
END_VAR
Serializer.AddReal(activeData);
END_METHOD

PROPERTY PUBLIC Size : UDINT
GET
Size := SIZEOF(activeData);
END_GET
END_PROPERTY

METHOD TryDeserializeFrom : BOOL
VAR_INPUT
	Deserializer : I_Deserializer;
	Feedback : I_DeserializerFeedback;
END_VAR
TryDeserializeFrom := Deserializer.TryGetReal(activeData, Feedback);
END_METHOD

METHOD TryMakeReferenceTo : BOOL
VAR_INPUT
	Target : I_Datatype;
END_VAR
VAR
	pTargetData : POINTER TO REAL;
END_VAR
IF NOT IsEquivalentTo(Target) THEN
	RETURN;
END_IF

pTargetData := Target.Address;
activeData REF= pTargetData^;
TryMakeReferenceTo := TRUE;
END_METHOD

PROPERTY PUBLIC TypeName : T_MAXSTRING
GET
TypeName := 'REAL';
END_GET
END_PROPERTY

PROPERTY PUBLIC Value : REFERENCE TO REAL
GET
Value REF= activeData;
END_GET
END_PROPERTY

END_FUNCTION_BLOCK

// mobject-converters/Converters/BOOL_TO_/TryConvert_BOOL_TO_LREAL
FUNCTION TryConvert_BOOL_TO_LREAL : BOOL
VAR_INPUT
	in : BOOL;
	out : REFERENCE TO LREAL;
END_VAR

out := BOOL_TO_LREAL(in);
TryConvert_BOOL_TO_LREAL := TRUE;

END_FUNCTION

// mobject-datatypes/Primitive/_LREAL
{attribute 'linkalways'} 
{attribute 'no_explicit_call' := 'This FB is a CLASS and must be accessed using methods or properties'}
{attribute 'enable_dynamic_creation'}
FUNCTION_BLOCK _LREAL EXTENDS NumericDatatypeBase
VAR
	localData : LREAL;
	activeData : REFERENCE TO LREAL REF= localData;
END_VAR

METHOD FB_init : BOOL
VAR_INPUT
	bInitRetains : BOOL; // if TRUE, the retain variables are initialized (warm start / cold start)
	bInCopyCode : BOOL;  // if TRUE, the instance afterwards gets moved into the copy code (online change)
	InitialValue : LREAL;
END_VAR
localData := InitialValue;
END_METHOD

METHOD PROTECTED SerializeMaxValue
VAR_INPUT
	Serializer : I_Serializer;
END_VAR
Serializer.AddLreal(MaxValue);
END_METHOD

METHOD PROTECTED SerializeMinValue
VAR_INPUT
	Serializer : I_Serializer;
END_VAR
Serializer.AddLreal(MinValue);
END_METHOD

PROPERTY PUBLIC Address : PVOID
GET
Address := ADR(activeData);
END_GET
END_PROPERTY

METHOD PUBLIC ClearReference
VAR_INPUT
END_VAR
activeData REF= localData;
END_METHOD

METHOD PUBLIC Clone : I_Datatype
VAR
    pClone : POINTER TO _LREAL;
END_VAR
pClone := __NEW(_LREAL(InitialValue := Value));
Clone := pClone^;
END_METHOD

PROPERTY PUBLIC IsEven : BOOL
GET
IsEven := FALSE;
END_GET
END_PROPERTY

PROPERTY PUBLIC IsFloat : BOOL
GET
IsFloat := TRUE;
END_GET
END_PROPERTY

PROPERTY PUBLIC IsOdd : BOOL
GET
IsOdd := FALSE;
END_GET
END_PROPERTY

PROPERTY PUBLIC IsSigned : BOOL
GET
IsSigned := TRUE;
END_GET
END_PROPERTY

METHOD PUBLIC MakeReferenceTo
VAR_INPUT
	ReferenceTarget : REFERENCE TO LREAL;
END_VAR
activeData REF= ReferenceTarget;
END_METHOD

PROPERTY PUBLIC MaxValue : LREAL
GET
MaxValue :=  DatatypeLimits.LREAL_MAX_VALUE;
END_GET
END_PROPERTY

PROPERTY PUBLIC MinValue : LREAL
GET
MinValue := DatatypeLimits.LREAL_MIN_VALUE;
END_GET
END_PROPERTY

METHOD PUBLIC SerializeWith
VAR_INPUT
	Serializer : I_Serializer;
END_VAR
Serializer.AddLreal(activeData);
END_METHOD

PROPERTY PUBLIC Size : UDINT
GET
Size := SIZEOF(activeData);
END_GET
END_PROPERTY

METHOD TryDeserializeFrom : BOOL
VAR_INPUT
	Deserializer : I_Deserializer;
	Feedback : I_DeserializerFeedback;
END_VAR
TryDeserializeFrom := Deserializer.TryGetLreal(activeData, Feedback);
END_METHOD

METHOD TryMakeReferenceTo : BOOL
VAR_INPUT
	Target : I_Datatype;
END_VAR
VAR
	pTargetData : POINTER TO LREAL;
END_VAR
IF NOT IsEquivalentTo(Target) THEN
	RETURN;
END_IF

pTargetData := Target.Address;
activeData REF= pTargetData^;
TryMakeReferenceTo := TRUE;
END_METHOD

PROPERTY PUBLIC TypeName : T_MAXSTRING
GET
TypeName := 'LREAL';
END_GET
END_PROPERTY

PROPERTY PUBLIC Value : REFERENCE TO LREAL
GET
Value REF= activeData;
END_GET
END_PROPERTY

END_FUNCTION_BLOCK

// mobject-converters/Converters/BOOL_TO_/TryConvert_BOOL_TO_TIME
FUNCTION TryConvert_BOOL_TO_TIME : BOOL
VAR_INPUT
	in : BOOL;
	out : REFERENCE TO TIME;
END_VAR

out := BOOL_TO_TIME(in);
TryConvert_BOOL_TO_TIME := TRUE;

END_FUNCTION

// mobject-converters/Converters/BOOL_TO_/TryConvert_BOOL_TO_TOD
FUNCTION TryConvert_BOOL_TO_TOD : BOOL
VAR_INPUT
	in : BOOL;
	out : REFERENCE TO TOD;
END_VAR

out := BOOL_TO_TOD(in);
TryConvert_BOOL_TO_TOD := TRUE;

END_FUNCTION

// mobject-datatypes/Primitive/_TOD
{attribute 'linkalways'} 
{attribute 'no_explicit_call' := 'This FB is a CLASS and must be accessed using methods or properties'}
{attribute 'enable_dynamic_creation'}
FUNCTION_BLOCK _TOD EXTENDS DatatypeBase
VAR
	localData : TOD;
	activeData : REFERENCE TO TOD REF= localData;
END_VAR

METHOD FB_init : BOOL
VAR_INPUT
	bInitRetains : BOOL; // if TRUE, the retain variables are initialized (warm start / cold start)
	bInCopyCode : BOOL;  // if TRUE, the instance afterwards gets moved WORDo the copy code (online change)
	InitialValue : TOD;
END_VAR
localData := InitialValue;
END_METHOD

PROPERTY PUBLIC Address : PVOID
GET
Address := ADR(activeData);
END_GET
END_PROPERTY

METHOD PUBLIC ClearReference
VAR_INPUT
END_VAR
activeData REF= localData;
END_METHOD

METHOD PUBLIC Clone : I_Datatype
VAR
    pClone : POINTER TO _TOD;
END_VAR
pClone := __NEW(_TOD(InitialValue := Value));
Clone := pClone^;
END_METHOD

METHOD PUBLIC MakeReferenceTo
VAR_INPUT
	ReferenceTarget : REFERENCE TO TOD;
END_VAR
activeData REF= ReferenceTarget;
END_METHOD

METHOD PUBLIC SerializeWith
VAR_INPUT
	Serializer : I_Serializer;
END_VAR
Serializer.AddTod(activeData);
END_METHOD

PROPERTY PUBLIC Size : UDINT
GET
Size := SIZEOF(activeData);
END_GET
END_PROPERTY

METHOD TryDeserializeFrom : BOOL
VAR_INPUT
	Deserializer : I_Deserializer;
	Feedback : I_DeserializerFeedback;
END_VAR
TryDeserializeFrom := Deserializer.TryGetTod(activeData, Feedback);
END_METHOD

METHOD TryMakeReferenceTo : BOOL
VAR_INPUT
	Target : I_Datatype;
END_VAR
VAR
	pTargetData : POINTER TO TOD;
END_VAR
IF NOT IsEquivalentTo(Target) THEN
	RETURN;
END_IF

pTargetData := Target.Address;
activeData REF= pTargetData^;
TryMakeReferenceTo := TRUE;
END_METHOD

PROPERTY PUBLIC TypeName : T_MAXSTRING
GET
TypeName := 'TOD';
END_GET
END_PROPERTY

PROPERTY PUBLIC Value : REFERENCE TO TOD
GET
Value REF= activeData;
END_GET
END_PROPERTY

END_FUNCTION_BLOCK

// mobject-converters/Converters/BOOL_TO_/TryConvert_BOOL_TO_DT
FUNCTION TryConvert_BOOL_TO_DT : BOOL
VAR_INPUT
	in : BOOL;
	out : REFERENCE TO DT;
END_VAR

out := BOOL_TO_DT(in);
TryConvert_BOOL_TO_DT := TRUE;

END_FUNCTION

// mobject-datatypes/Primitive/_DT
{attribute 'linkalways'} 
{attribute 'no_explicit_call' := 'This FB is a CLASS and must be accessed using methods or properties'}
{attribute 'enable_dynamic_creation'}
FUNCTION_BLOCK _DT EXTENDS DatatypeBase
VAR
	localData : DT;
	activeData : REFERENCE TO DT REF= localData;
END_VAR

METHOD FB_init : BOOL
VAR_INPUT
	bInitRetains : BOOL; // if TRUE, the retain variables are initialized (warm start / cold start)
	bInCopyCode : BOOL;  // if TRUE, the instance afterwards gets moved WORDo the copy code (online change)
	InitialValue : DT;
END_VAR
localData := InitialValue;
END_METHOD

PROPERTY PUBLIC Address : PVOID
GET
Address := ADR(activeData);
END_GET
END_PROPERTY

METHOD PUBLIC ClearReference
VAR_INPUT
END_VAR
activeData REF= localData;
END_METHOD

METHOD PUBLIC Clone : I_Datatype
VAR
    pClone : POINTER TO _DT;
END_VAR
pClone := __NEW(_DT(InitialValue := Value));
Clone := pClone^;
END_METHOD

METHOD PUBLIC MakeReferenceTo
VAR_INPUT
	ReferenceTarget : REFERENCE TO DT;
END_VAR
activeData REF= ReferenceTarget;
END_METHOD

METHOD PUBLIC SerializeWith
VAR_INPUT
	Serializer : I_Serializer;
END_VAR
Serializer.AddDateTime(activeData);
END_METHOD

PROPERTY PUBLIC Size : UDINT
GET
Size := SIZEOF(activeData);
END_GET
END_PROPERTY

METHOD TryDeserializeFrom : BOOL
VAR_INPUT
	Deserializer : I_Deserializer;
	Feedback : I_DeserializerFeedback;
END_VAR
TryDeserializeFrom := Deserializer.TryGetDateTime(activeData, Feedback);
END_METHOD

METHOD TryMakeReferenceTo : BOOL
VAR_INPUT
	Target : I_Datatype;
END_VAR
VAR
	pTargetData : POINTER TO DT;
END_VAR
IF NOT IsEquivalentTo(Target) THEN
	RETURN;
END_IF

pTargetData := Target.Address;
activeData REF= pTargetData^;
TryMakeReferenceTo := TRUE;
END_METHOD

PROPERTY PUBLIC TypeName : T_MAXSTRING
GET
TypeName := 'DT';
END_GET
END_PROPERTY

PROPERTY PUBLIC Value : REFERENCE TO DT
GET
Value REF= activeData;
END_GET
END_PROPERTY

END_FUNCTION_BLOCK

// mobject-converters/Converters/BOOL_TO_/TryConvert_BOOL_TO_STRING
FUNCTION TryConvert_BOOL_TO_STRING : BOOL
VAR_INPUT
	in : BOOL;
	out : REFERENCE TO STRING;
END_VAR

out := BOOL_TO_STRING(in);
TryConvert_BOOL_TO_STRING := TRUE;

END_FUNCTION

// mobject-datatypes/Primitive/_STRING
{attribute 'linkalways'} 
{attribute 'no_explicit_call' := 'This FB is a CLASS and must be accessed using methods or properties'}
{attribute 'enable_dynamic_creation'}
FUNCTION_BLOCK _STRING EXTENDS DatatypeBase
VAR
	localData : T_MaxString;
	activeData : REFERENCE TO T_MaxString REF= localData;
END_VAR

METHOD FB_init : BOOL
VAR_INPUT
	bInitRetains : BOOL; // if TRUE, the retain variables are initialized (warm start / cold start)
	bInCopyCode : BOOL;  // if TRUE, the instance afterwards gets moved WORDo the copy code (online change)
	InitialValue : T_MaxString;
END_VAR
localData := InitialValue;
END_METHOD

PROPERTY PUBLIC Address : PVOID
GET
Address := ADR(activeData);
END_GET
END_PROPERTY

METHOD PUBLIC ClearReference
VAR_INPUT
END_VAR
activeData REF= localData;
END_METHOD

METHOD PUBLIC Clone : I_Datatype
VAR
    pClone : POINTER TO _STRING;
END_VAR
pClone := __NEW(_STRING(InitialValue := Value));
Clone := pClone^;
END_METHOD

PROPERTY PUBLIC Length : INT
GET
Length := len(activeData);
END_GET
END_PROPERTY

METHOD PUBLIC MakeReferenceTo
VAR_INPUT
	ReferenceTarget : REFERENCE TO T_MaxString;
END_VAR
activeData REF= ReferenceTarget;
END_METHOD

METHOD PUBLIC SerializeWith
VAR_INPUT
	Serializer : I_Serializer;
END_VAR
Serializer.AddString(activeData);
END_METHOD

PROPERTY PUBLIC Size : UDINT
GET
Size := SIZEOF(activeData);
END_GET
END_PROPERTY

METHOD TryDeserializeFrom : BOOL
VAR_INPUT
	Deserializer : I_Deserializer;
	Feedback : I_DeserializerFeedback;
END_VAR
TryDeserializeFrom := Deserializer.TryGetString(activeData, Feedback);
END_METHOD

METHOD TryMakeReferenceTo : BOOL
VAR_INPUT
	Target : I_Datatype;
END_VAR
VAR
	pTargetData : POINTER TO T_MaxString;
END_VAR
IF NOT IsEquivalentTo(Target) THEN
	RETURN;
END_IF

pTargetData := Target.Address;
activeData REF= pTargetData^;
TryMakeReferenceTo := TRUE;
END_METHOD

PROPERTY PUBLIC TypeName : T_MAXSTRING
GET
TypeName := 'STRING';
END_GET
END_PROPERTY

PROPERTY PUBLIC Value : REFERENCE TO T_MaxString
GET
Value REF= activeData;
END_GET
END_PROPERTY

END_FUNCTION_BLOCK

// mobject-converters/Converters/BYTE_TO_/TryConvert_BYTE_TO_BOOL
FUNCTION TryConvert_BYTE_TO_BOOL : BOOL
VAR_INPUT
	in : BYTE;
	out : REFERENCE TO BOOL;
END_VAR

out := BYTE_TO_BOOL(in);
TryConvert_BYTE_TO_BOOL := TRUE;

END_FUNCTION

// mobject-converters/Converters/BYTE_TO_/TryConvert_BYTE_TO_BYTE
FUNCTION TryConvert_BYTE_TO_BYTE : BOOL
VAR_INPUT
	in : BYTE;
	out : REFERENCE TO BYTE;
END_VAR

out := in;
TryConvert_BYTE_TO_BYTE := TRUE;

END_FUNCTION

// mobject-converters/Converters/BYTE_TO_/TryConvert_BYTE_TO_DATE
FUNCTION TryConvert_BYTE_TO_DATE : BOOL
VAR_INPUT
	in : BYTE;
	out : REFERENCE TO DATE;
END_VAR

out := BYTE_TO_DATE(in);
TryConvert_BYTE_TO_DATE := TRUE;

END_FUNCTION

// mobject-converters/Converters/BYTE_TO_/TryConvert_BYTE_TO_Destination
FUNCTION TryConvert_BYTE_TO_Destination : BOOL
VAR_INPUT
	in : BYTE;
	out : ANY;
END_VAR
VAR
	convertResult : BOOL := FALSE;
	convertAddress : PVOID;
	_BOOL : BOOL;
	_BYTE : BYTE;
	_WORD : WORD;
	_DWORD : DWORD;
	_LWORD : LWORD;
	_SINT : SINT;
	_INT : INT;
	_DINT : DINT;
	_LINT : LINT;
	_USINT : USINT;
	_UINT : UINT;
	_UDINT : UDINT;
	_ULINT : ULINT;
	_REAL : REAL;
	_LREAL : LREAL;
	_TIME : TIME;
	_TOD : TOD;
	_DATE : DATE;
	_DT : DT;
	_STRING : STRING;
END_VAR

CASE out.TypeClass OF
	__SYSTEM.TYPE_CLASS.TYPE_BOOL:
	
	convertResult := TryConvert_BYTE_TO_BOOL(in, _BOOL);
	IF convertResult THEN
		convertAddress := ADR(_BOOL);
	END_IF
	
	__SYSTEM.TYPE_CLASS.TYPE_BYTE:
	
	convertResult := TryConvert_BYTE_TO_BYTE(in, _BYTE);
	IF convertResult THEN
		convertAddress := ADR(_BYTE);
	END_IF
	
	__SYSTEM.TYPE_CLASS.TYPE_WORD:
	
	convertResult := TryConvert_BYTE_TO_WORD(in, _WORD);
	IF convertResult THEN
		convertAddress := ADR(_WORD);
	END_IF
	
	__SYSTEM.TYPE_CLASS.TYPE_DWORD:
	
	convertResult := TryConvert_BYTE_TO_DWORD(in, _DWORD);
	IF convertResult THEN
		convertAddress := ADR(_DWORD);
	END_IF
	
	__SYSTEM.TYPE_CLASS.TYPE_LWORD:
	
	convertResult := TryConvert_BYTE_TO_LWORD(in, _LWORD);
	IF convertResult THEN
		convertAddress := ADR(_LWORD);
	END_IF
	
	__SYSTEM.TYPE_CLASS.TYPE_SINT:
	
	convertResult := TryConvert_BYTE_TO_SINT(in, _SINT);
	IF convertResult THEN
		convertAddress := ADR(_SINT);
	END_IF
	
	__SYSTEM.TYPE_CLASS.TYPE_INT:
	
	convertResult := TryConvert_BYTE_TO_INT(in, _INT);
	IF convertResult THEN
		convertAddress := ADR(_INT);
	END_IF
	
	__SYSTEM.TYPE_CLASS.TYPE_DINT:
	
	convertResult := TryConvert_BYTE_TO_DINT(in, _DINT);
	IF convertResult THEN
		convertAddress := ADR(_DINT);
	END_IF
	
	__SYSTEM.TYPE_CLASS.TYPE_LINT:
	
	convertResult := TryConvert_BYTE_TO_LINT(in, _LINT);
	IF convertResult THEN
		convertAddress := ADR(_LINT);
	END_IF
	
	__SYSTEM.TYPE_CLASS.TYPE_USINT:
	
	convertResult := TryConvert_BYTE_TO_USINT(in, _USINT);
	IF convertResult THEN
		convertAddress := ADR(_USINT);
	END_IF
	
	__SYSTEM.TYPE_CLASS.TYPE_UINT:
	
	convertResult := TryConvert_BYTE_TO_UINT(in, _UINT);
	IF convertResult THEN
		convertAddress := ADR(_UINT);
	END_IF
	
	__SYSTEM.TYPE_CLASS.TYPE_UDINT:
	
	convertResult := TryConvert_BYTE_TO_UDINT(in, _UDINT);
	IF convertResult THEN
		convertAddress := ADR(_UDINT);
	END_IF
	
	__SYSTEM.TYPE_CLASS.TYPE_ULINT:
	
	convertResult := TryConvert_BYTE_TO_ULINT(in, _ULINT);
	IF convertResult THEN
		convertAddress := ADR(_ULINT);
	END_IF
	
	__SYSTEM.TYPE_CLASS.TYPE_REAL:
	
	convertResult := TryConvert_BYTE_TO_REAL(in, _REAL);
	IF convertResult THEN
		convertAddress := ADR(_REAL);
	END_IF
	
	__SYSTEM.TYPE_CLASS.TYPE_LREAL:
	
	convertResult := TryConvert_BYTE_TO_LREAL(in, _LREAL);
	IF convertResult THEN
		convertAddress := ADR(_LREAL);
	END_IF
	
	__SYSTEM.TYPE_CLASS.TYPE_TIME:
	
	convertResult := TryConvert_BYTE_TO_TIME(in, _TIME);
	IF convertResult THEN
		convertAddress := ADR(_TIME);
	END_IF
	
	__SYSTEM.TYPE_CLASS.TYPE_TIMEOFDAY:
	
	convertResult := TryConvert_BYTE_TO_TOD(in, _TOD);
	IF convertResult THEN
		convertAddress := ADR(_TOD);
	END_IF
	
	__SYSTEM.TYPE_CLASS.TYPE_DATE:
	
	convertResult := TryConvert_BYTE_TO_DATE(in, _DATE);
	IF convertResult THEN
		convertAddress := ADR(_DATE);
	END_IF
	
	__SYSTEM.TYPE_CLASS.TYPE_DATEANDTIME:
	
	convertResult := TryConvert_BYTE_TO_DT(in, _DT);
	IF convertResult THEN
		convertAddress := ADR(_DT);
	END_IF
	
	__SYSTEM.TYPE_CLASS.TYPE_STRING:
	
	convertResult := TryConvert_BYTE_TO_STRING(in, _STRING);
	IF convertResult THEN
		convertAddress := ADR(_STRING);
	END_IF
	
END_CASE

IF convertResult THEN
	memcpy(out.pValue,convertAddress,DINT_TO_UDINT(out.diSize));
END_IF

TryConvert_BYTE_TO_Destination := convertResult;

END_FUNCTION

// mobject-converters/Converters/BYTE_TO_/TryConvert_BYTE_TO_WORD
FUNCTION TryConvert_BYTE_TO_WORD : BOOL
VAR_INPUT
	in : BYTE;
	out : REFERENCE TO WORD;
END_VAR

out := BYTE_TO_WORD(in);
TryConvert_BYTE_TO_WORD := TRUE;

END_FUNCTION

// mobject-converters/Converters/BYTE_TO_/TryConvert_BYTE_TO_DWORD
FUNCTION TryConvert_BYTE_TO_DWORD : BOOL
VAR_INPUT
	in : BYTE;
	out : REFERENCE TO DWORD;
END_VAR

out := BYTE_TO_DWORD(in);
TryConvert_BYTE_TO_DWORD := TRUE;

END_FUNCTION

// mobject-converters/Converters/BYTE_TO_/TryConvert_BYTE_TO_LWORD
FUNCTION TryConvert_BYTE_TO_LWORD : BOOL
VAR_INPUT
	in : BYTE;
	out : REFERENCE TO LWORD;
END_VAR

out := BYTE_TO_LWORD(in);
TryConvert_BYTE_TO_LWORD := TRUE;

END_FUNCTION

// mobject-converters/Converters/BYTE_TO_/TryConvert_BYTE_TO_SINT
FUNCTION TryConvert_BYTE_TO_SINT : BOOL
VAR_INPUT
	in : BYTE;
	out : REFERENCE TO SINT;
END_VAR

IF in > DatatypeLimits.MAX_VALUE_OF_BYTE_WHICH_CAN_BE_HELD_IN_A_SINT THEN
	RETURN;
END_IF

out := BYTE_TO_SINT(in);
TryConvert_BYTE_TO_SINT := TRUE;

END_FUNCTION

// mobject-converters/Converters/BYTE_TO_/TryConvert_BYTE_TO_INT
FUNCTION TryConvert_BYTE_TO_INT : BOOL
VAR_INPUT
	in : BYTE;
	out : REFERENCE TO INT;
END_VAR

out := BYTE_TO_INT(in);
TryConvert_BYTE_TO_INT := TRUE;

END_FUNCTION

// mobject-converters/Converters/BYTE_TO_/TryConvert_BYTE_TO_DINT
FUNCTION TryConvert_BYTE_TO_DINT : BOOL
VAR_INPUT
	in : BYTE;
	out : REFERENCE TO DINT;
END_VAR

out := BYTE_TO_DINT(in);
TryConvert_BYTE_TO_DINT := TRUE;

END_FUNCTION

// mobject-converters/Converters/BYTE_TO_/TryConvert_BYTE_TO_LINT
FUNCTION TryConvert_BYTE_TO_LINT : BOOL
VAR_INPUT
	in : BYTE;
	out : REFERENCE TO LINT;
END_VAR

out := BYTE_TO_LINT(in);
TryConvert_BYTE_TO_LINT := TRUE;

END_FUNCTION

// mobject-converters/Converters/BYTE_TO_/TryConvert_BYTE_TO_USINT
FUNCTION TryConvert_BYTE_TO_USINT : BOOL
VAR_INPUT
	in : BYTE;
	out : REFERENCE TO USINT;
END_VAR

out := BYTE_TO_USINT(in);
TryConvert_BYTE_TO_USINT := TRUE;

END_FUNCTION

// mobject-converters/Converters/BYTE_TO_/TryConvert_BYTE_TO_UINT
FUNCTION TryConvert_BYTE_TO_UINT : BOOL
VAR_INPUT
	in : BYTE;
	out : REFERENCE TO UINT;
END_VAR

out := BYTE_TO_UINT(in);
TryConvert_BYTE_TO_UINT := TRUE;

END_FUNCTION

// mobject-converters/Converters/BYTE_TO_/TryConvert_BYTE_TO_UDINT
FUNCTION TryConvert_BYTE_TO_UDINT : BOOL
VAR_INPUT
	in : BYTE;
	out : REFERENCE TO UDINT;
END_VAR

out := BYTE_TO_UDINT(in);
TryConvert_BYTE_TO_UDINT := TRUE;

END_FUNCTION

// mobject-converters/Converters/BYTE_TO_/TryConvert_BYTE_TO_ULINT
FUNCTION TryConvert_BYTE_TO_ULINT : BOOL
VAR_INPUT
	in : BYTE;
	out : REFERENCE TO ULINT;
END_VAR

out := BYTE_TO_ULINT(in);
TryConvert_BYTE_TO_ULINT := TRUE;

END_FUNCTION

// mobject-converters/Converters/BYTE_TO_/TryConvert_BYTE_TO_REAL
FUNCTION TryConvert_BYTE_TO_REAL : BOOL
VAR_INPUT
	in : BYTE;
	out : REFERENCE TO REAL;
END_VAR

out := BYTE_TO_REAL(in);
TryConvert_BYTE_TO_REAL := TRUE;

END_FUNCTION

// mobject-converters/Converters/BYTE_TO_/TryConvert_BYTE_TO_LREAL
FUNCTION TryConvert_BYTE_TO_LREAL : BOOL
VAR_INPUT
	in : BYTE;
	out : REFERENCE TO LREAL;
END_VAR

out := BYTE_TO_LREAL(in);
TryConvert_BYTE_TO_LREAL := TRUE;

END_FUNCTION

// mobject-converters/Converters/BYTE_TO_/TryConvert_BYTE_TO_TIME
FUNCTION TryConvert_BYTE_TO_TIME : BOOL
VAR_INPUT
	in : BYTE;
	out : REFERENCE TO TIME;
END_VAR

out := BYTE_TO_TIME(in);
TryConvert_BYTE_TO_TIME := TRUE;

END_FUNCTION

// mobject-converters/Converters/BYTE_TO_/TryConvert_BYTE_TO_TOD
FUNCTION TryConvert_BYTE_TO_TOD : BOOL
VAR_INPUT
	in : BYTE;
	out : REFERENCE TO TOD;
END_VAR

out := BYTE_TO_TOD(in);
TryConvert_BYTE_TO_TOD := TRUE;

END_FUNCTION

// mobject-converters/Converters/BYTE_TO_/TryConvert_BYTE_TO_DT
FUNCTION TryConvert_BYTE_TO_DT : BOOL
VAR_INPUT
	in : BYTE;
	out : REFERENCE TO DT;
END_VAR

out := BYTE_TO_DT(in);
TryConvert_BYTE_TO_DT := TRUE;

END_FUNCTION

// mobject-converters/Converters/BYTE_TO_/TryConvert_BYTE_TO_STRING
FUNCTION TryConvert_BYTE_TO_STRING : BOOL
VAR_INPUT
	in : BYTE;
	out : REFERENCE TO STRING;
END_VAR

out := BYTE_TO_STRING(in);
TryConvert_BYTE_TO_STRING := TRUE;

END_FUNCTION

// mobject-converters/Converters/DATE_TO_/TryConvert_DATE_TO_BOOL
FUNCTION TryConvert_DATE_TO_BOOL : BOOL
VAR_INPUT
	in : DATE;
	out : REFERENCE TO BOOL;
END_VAR

out := DATE_TO_BOOL(in);
TryConvert_DATE_TO_BOOL := TRUE;

END_FUNCTION

// mobject-converters/Converters/DATE_TO_/TryConvert_DATE_TO_BYTE
FUNCTION TryConvert_DATE_TO_BYTE : BOOL
VAR_INPUT
	in : DATE;
	out : REFERENCE TO BYTE;
END_VAR

IF in > DatatypeLimits.MAX_VALUE_OF_DATE_WHICH_CAN_BE_HELD_IN_A_BYTE THEN
	RETURN;
END_IF

out := DATE_TO_BYTE(in);
TryConvert_DATE_TO_BYTE := TRUE;

END_FUNCTION

// mobject-converters/Converters/DATE_TO_/TryConvert_DATE_TO_DATE
FUNCTION TryConvert_DATE_TO_DATE : BOOL
VAR_INPUT
	in : DATE;
	out : REFERENCE TO DATE;
END_VAR

out := in;
TryConvert_DATE_TO_DATE := TRUE;

END_FUNCTION

// mobject-converters/Converters/DATE_TO_/TryConvert_DATE_TO_Destination
FUNCTION TryConvert_DATE_TO_Destination : BOOL
VAR_INPUT
	in : DATE;
	out : ANY;
END_VAR
VAR
	convertResult : BOOL := FALSE;
	convertAddress : PVOID;
	_BOOL : BOOL;
	_BYTE : BYTE;
	_WORD : WORD;
	_DWORD : DWORD;
	_LWORD : LWORD;
	_SINT : SINT;
	_INT : INT;
	_DINT : DINT;
	_LINT : LINT;
	_USINT : USINT;
	_UINT : UINT;
	_UDINT : UDINT;
	_ULINT : ULINT;
	_REAL : REAL;
	_LREAL : LREAL;
	_TIME : TIME;
	_TOD : TOD;
	_DATE : DATE;
	_DT : DT;
	_STRING : STRING;
END_VAR

CASE out.TypeClass OF
	__SYSTEM.TYPE_CLASS.TYPE_BOOL:
	
	convertResult := TryConvert_DATE_TO_BOOL(in, _BOOL);
	IF convertResult THEN
		convertAddress := ADR(_BOOL);
	END_IF
	
	__SYSTEM.TYPE_CLASS.TYPE_BYTE:
	
	convertResult := TryConvert_DATE_TO_BYTE(in, _BYTE);
	IF convertResult THEN
		convertAddress := ADR(_BYTE);
	END_IF
	
	__SYSTEM.TYPE_CLASS.TYPE_WORD:
	
	convertResult := TryConvert_DATE_TO_WORD(in, _WORD);
	IF convertResult THEN
		convertAddress := ADR(_WORD);
	END_IF
	
	__SYSTEM.TYPE_CLASS.TYPE_DWORD:
	
	convertResult := TryConvert_DATE_TO_DWORD(in, _DWORD);
	IF convertResult THEN
		convertAddress := ADR(_DWORD);
	END_IF
	
	__SYSTEM.TYPE_CLASS.TYPE_LWORD:
	
	convertResult := TryConvert_DATE_TO_LWORD(in, _LWORD);
	IF convertResult THEN
		convertAddress := ADR(_LWORD);
	END_IF
	
	__SYSTEM.TYPE_CLASS.TYPE_SINT:
	
	convertResult := TryConvert_DATE_TO_SINT(in, _SINT);
	IF convertResult THEN
		convertAddress := ADR(_SINT);
	END_IF
	
	__SYSTEM.TYPE_CLASS.TYPE_INT:
	
	convertResult := TryConvert_DATE_TO_INT(in, _INT);
	IF convertResult THEN
		convertAddress := ADR(_INT);
	END_IF
	
	__SYSTEM.TYPE_CLASS.TYPE_DINT:
	
	convertResult := TryConvert_DATE_TO_DINT(in, _DINT);
	IF convertResult THEN
		convertAddress := ADR(_DINT);
	END_IF
	
	__SYSTEM.TYPE_CLASS.TYPE_LINT:
	
	convertResult := TryConvert_DATE_TO_LINT(in, _LINT);
	IF convertResult THEN
		convertAddress := ADR(_LINT);
	END_IF
	
	__SYSTEM.TYPE_CLASS.TYPE_USINT:
	
	convertResult := TryConvert_DATE_TO_USINT(in, _USINT);
	IF convertResult THEN
		convertAddress := ADR(_USINT);
	END_IF
	
	__SYSTEM.TYPE_CLASS.TYPE_UINT:
	
	convertResult := TryConvert_DATE_TO_UINT(in, _UINT);
	IF convertResult THEN
		convertAddress := ADR(_UINT);
	END_IF
	
	__SYSTEM.TYPE_CLASS.TYPE_UDINT:
	
	convertResult := TryConvert_DATE_TO_UDINT(in, _UDINT);
	IF convertResult THEN
		convertAddress := ADR(_UDINT);
	END_IF
	
	__SYSTEM.TYPE_CLASS.TYPE_ULINT:
	
	convertResult := TryConvert_DATE_TO_ULINT(in, _ULINT);
	IF convertResult THEN
		convertAddress := ADR(_ULINT);
	END_IF
	
	__SYSTEM.TYPE_CLASS.TYPE_REAL:
	
	convertResult := TryConvert_DATE_TO_REAL(in, _REAL);
	IF convertResult THEN
		convertAddress := ADR(_REAL);
	END_IF
	
	__SYSTEM.TYPE_CLASS.TYPE_LREAL:
	
	convertResult := TryConvert_DATE_TO_LREAL(in, _LREAL);
	IF convertResult THEN
		convertAddress := ADR(_LREAL);
	END_IF
	
	__SYSTEM.TYPE_CLASS.TYPE_TIME:
	
	convertResult := TryConvert_DATE_TO_TIME(in, _TIME);
	IF convertResult THEN
		convertAddress := ADR(_TIME);
	END_IF
	
	__SYSTEM.TYPE_CLASS.TYPE_TIMEOFDAY:
	
	convertResult := TryConvert_DATE_TO_TOD(in, _TOD);
	IF convertResult THEN
		convertAddress := ADR(_TOD);
	END_IF
	
	__SYSTEM.TYPE_CLASS.TYPE_DATE:
	
	convertResult := TryConvert_DATE_TO_DATE(in, _DATE);
	IF convertResult THEN
		convertAddress := ADR(_DATE);
	END_IF
	
	__SYSTEM.TYPE_CLASS.TYPE_DATEANDTIME:
	
	convertResult := TryConvert_DATE_TO_DT(in, _DT);
	IF convertResult THEN
		convertAddress := ADR(_DT);
	END_IF
	
	__SYSTEM.TYPE_CLASS.TYPE_STRING:
	
	convertResult := TryConvert_DATE_TO_STRING(in, _STRING);
	IF convertResult THEN
		convertAddress := ADR(_STRING);
	END_IF
	
END_CASE

IF convertResult THEN
	memcpy(out.pValue,convertAddress,DINT_TO_UDINT(out.diSize));
END_IF

TryConvert_DATE_TO_Destination := convertResult;

END_FUNCTION

// mobject-converters/Converters/DATE_TO_/TryConvert_DATE_TO_WORD
FUNCTION TryConvert_DATE_TO_WORD : BOOL
VAR_INPUT
	in : DATE;
	out : REFERENCE TO WORD;
END_VAR

IF in > DatatypeLimits.MAX_VALUE_OF_DATE_WHICH_CAN_BE_HELD_IN_A_WORD THEN
	RETURN;
END_IF

out := DATE_TO_WORD(in);
TryConvert_DATE_TO_WORD := TRUE;

END_FUNCTION

// mobject-converters/Converters/DATE_TO_/TryConvert_DATE_TO_DWORD
FUNCTION TryConvert_DATE_TO_DWORD : BOOL
VAR_INPUT
	in : DATE;
	out : REFERENCE TO DWORD;
END_VAR

out := DATE_TO_DWORD(in);
TryConvert_DATE_TO_DWORD := TRUE;

END_FUNCTION

// mobject-converters/Converters/DATE_TO_/TryConvert_DATE_TO_LWORD
FUNCTION TryConvert_DATE_TO_LWORD : BOOL
VAR_INPUT
	in : DATE;
	out : REFERENCE TO LWORD;
END_VAR

out := DATE_TO_LWORD(in);
TryConvert_DATE_TO_LWORD := TRUE;

END_FUNCTION

// mobject-converters/Converters/DATE_TO_/TryConvert_DATE_TO_SINT
FUNCTION TryConvert_DATE_TO_SINT : BOOL
VAR_INPUT
	in : DATE;
	out : REFERENCE TO SINT;
END_VAR

IF in > DatatypeLimits.MAX_VALUE_OF_DATE_WHICH_CAN_BE_HELD_IN_A_SINT THEN
	RETURN;
END_IF

out := DATE_TO_SINT(in);
TryConvert_DATE_TO_SINT := TRUE;

END_FUNCTION

// mobject-converters/Converters/DATE_TO_/TryConvert_DATE_TO_INT
FUNCTION TryConvert_DATE_TO_INT : BOOL
VAR_INPUT
	in : DATE;
	out : REFERENCE TO INT;
END_VAR

IF in > DatatypeLimits.MAX_VALUE_OF_DATE_WHICH_CAN_BE_HELD_IN_A_INT THEN
	RETURN;
END_IF

out := DATE_TO_INT(in);
TryConvert_DATE_TO_INT := TRUE;

END_FUNCTION

// mobject-converters/Converters/DATE_TO_/TryConvert_DATE_TO_DINT
FUNCTION TryConvert_DATE_TO_DINT : BOOL
VAR_INPUT
	in : DATE;
	out : REFERENCE TO DINT;
END_VAR

IF in > DatatypeLimits.MAX_VALUE_OF_DATE_WHICH_CAN_BE_HELD_IN_A_DINT THEN
	RETURN;
END_IF

out := DATE_TO_DINT(in);
TryConvert_DATE_TO_DINT := TRUE;

END_FUNCTION

// mobject-converters/Converters/DATE_TO_/TryConvert_DATE_TO_LINT
FUNCTION TryConvert_DATE_TO_LINT : BOOL
VAR_INPUT
	in : DATE;
	out : REFERENCE TO LINT;
END_VAR

out := DATE_TO_LINT(in);
TryConvert_DATE_TO_LINT := TRUE;

END_FUNCTION

// mobject-converters/Converters/DATE_TO_/TryConvert_DATE_TO_USINT
FUNCTION TryConvert_DATE_TO_USINT : BOOL
VAR_INPUT
	in : DATE;
	out : REFERENCE TO USINT;
END_VAR

IF in > DatatypeLimits.MAX_VALUE_OF_DATE_WHICH_CAN_BE_HELD_IN_A_USINT THEN
	RETURN;
END_IF

out := DATE_TO_USINT(in);
TryConvert_DATE_TO_USINT := TRUE;

END_FUNCTION

// mobject-converters/Converters/DATE_TO_/TryConvert_DATE_TO_UINT
FUNCTION TryConvert_DATE_TO_UINT : BOOL
VAR_INPUT
	in : DATE;
	out : REFERENCE TO UINT;
END_VAR

IF in > DatatypeLimits.MAX_VALUE_OF_DATE_WHICH_CAN_BE_HELD_IN_A_UINT THEN
	RETURN;
END_IF

out := DATE_TO_UINT(in);
TryConvert_DATE_TO_UINT := TRUE;

END_FUNCTION

// mobject-converters/Converters/DATE_TO_/TryConvert_DATE_TO_UDINT
FUNCTION TryConvert_DATE_TO_UDINT : BOOL
VAR_INPUT
	in : DATE;
	out : REFERENCE TO UDINT;
END_VAR

out := DATE_TO_UDINT(in);
TryConvert_DATE_TO_UDINT := TRUE;

END_FUNCTION

// mobject-converters/Converters/DATE_TO_/TryConvert_DATE_TO_ULINT
FUNCTION TryConvert_DATE_TO_ULINT : BOOL
VAR_INPUT
	in : DATE;
	out : REFERENCE TO ULINT;
END_VAR

out := DATE_TO_ULINT(in);
TryConvert_DATE_TO_ULINT := TRUE;

END_FUNCTION

// mobject-converters/Converters/DATE_TO_/TryConvert_DATE_TO_REAL
FUNCTION TryConvert_DATE_TO_REAL : BOOL
VAR_INPUT
	in : DATE;
	out : REFERENCE TO REAL;
END_VAR

out := DATE_TO_REAL(in);
TryConvert_DATE_TO_REAL := TRUE;

END_FUNCTION

// mobject-converters/Converters/DATE_TO_/TryConvert_DATE_TO_LREAL
FUNCTION TryConvert_DATE_TO_LREAL : BOOL
VAR_INPUT
	in : DATE;
	out : REFERENCE TO LREAL;
END_VAR

out := DATE_TO_LREAL(in);
TryConvert_DATE_TO_LREAL := TRUE;

END_FUNCTION

// mobject-converters/Converters/DATE_TO_/TryConvert_DATE_TO_TIME
FUNCTION TryConvert_DATE_TO_TIME : BOOL
VAR_INPUT
	in : DATE;
	out : REFERENCE TO TIME;
END_VAR

IF in > DatatypeLimits.MAX_VALUE_OF_DATE_WHICH_CAN_BE_HELD_IN_A_TIME THEN
	RETURN;
END_IF

out := DATE_TO_TIME(in);
TryConvert_DATE_TO_TIME := TRUE;

END_FUNCTION

// mobject-converters/Converters/DATE_TO_/TryConvert_DATE_TO_TOD
FUNCTION TryConvert_DATE_TO_TOD : BOOL
VAR_INPUT
	in : DATE;
	out : REFERENCE TO TOD;
END_VAR

IF in > DatatypeLimits.MAX_VALUE_OF_DATE_WHICH_CAN_BE_HELD_IN_A_TOD THEN
	RETURN;
END_IF

out := DATE_TO_TOD(in);
TryConvert_DATE_TO_TOD := TRUE;

END_FUNCTION

// mobject-converters/Converters/DATE_TO_/TryConvert_DATE_TO_DT
FUNCTION TryConvert_DATE_TO_DT : BOOL
VAR_INPUT
	in : DATE;
	out : REFERENCE TO DT;
END_VAR

IF in > DatatypeLimits.MAX_VALUE_OF_DATE_WHICH_CAN_BE_HELD_IN_A_DT THEN
	RETURN;
END_IF

out := DATE_TO_DT(in);
TryConvert_DATE_TO_DT := TRUE;

END_FUNCTION

// mobject-converters/Converters/DATE_TO_/TryConvert_DATE_TO_STRING
FUNCTION TryConvert_DATE_TO_STRING : BOOL
VAR_INPUT
	in : DATE;
	out : REFERENCE TO STRING;
END_VAR

out := DATE_TO_STRING(in);
TryConvert_DATE_TO_STRING := TRUE;

END_FUNCTION

// mobject-converters/Converters/DINT_TO_/TryConvert_DINT_TO_BOOL
FUNCTION TryConvert_DINT_TO_BOOL : BOOL
VAR_INPUT
	in : DINT;
	out : REFERENCE TO BOOL;
END_VAR

out := DINT_TO_BOOL(in);
TryConvert_DINT_TO_BOOL := TRUE;

END_FUNCTION

// mobject-converters/Converters/DINT_TO_/TryConvert_DINT_TO_BYTE
FUNCTION TryConvert_DINT_TO_BYTE : BOOL
VAR_INPUT
	in : DINT;
	out : REFERENCE TO BYTE;
END_VAR

IF in > DatatypeLimits.MAX_VALUE_OF_DINT_WHICH_CAN_BE_HELD_IN_A_BYTE THEN
	RETURN;
END_IF

IF in < DatatypeLimits.MIN_VALUE_OF_DINT_WHICH_CAN_BE_HELD_IN_A_BYTE THEN
	RETURN;
END_IF

out := DINT_TO_BYTE(in);
TryConvert_DINT_TO_BYTE := TRUE;

END_FUNCTION

// mobject-converters/Converters/DINT_TO_/TryConvert_DINT_TO_DATE
FUNCTION TryConvert_DINT_TO_DATE : BOOL
VAR_INPUT
	in : DINT;
	out : REFERENCE TO DATE;
END_VAR

IF in < DatatypeLimits.MIN_VALUE_OF_DINT_WHICH_CAN_BE_HELD_IN_A_DATE THEN
	RETURN;
END_IF

out := DINT_TO_DATE(in);
TryConvert_DINT_TO_DATE := TRUE;

END_FUNCTION

// mobject-converters/Converters/DINT_TO_/TryConvert_DINT_TO_Destination
FUNCTION TryConvert_DINT_TO_Destination : BOOL
VAR_INPUT
	in : DINT;
	out : ANY;
END_VAR
VAR
	convertResult : BOOL := FALSE;
	convertAddress : PVOID;
	_BOOL : BOOL;
	_BYTE : BYTE;
	_WORD : WORD;
	_DWORD : DWORD;
	_LWORD : LWORD;
	_SINT : SINT;
	_INT : INT;
	_DINT : DINT;
	_LINT : LINT;
	_USINT : USINT;
	_UINT : UINT;
	_UDINT : UDINT;
	_ULINT : ULINT;
	_REAL : REAL;
	_LREAL : LREAL;
	_TIME : TIME;
	_TOD : TOD;
	_DATE : DATE;
	_DT : DT;
	_STRING : STRING;
END_VAR

CASE out.TypeClass OF
	__SYSTEM.TYPE_CLASS.TYPE_BOOL:
	
	convertResult := TryConvert_DINT_TO_BOOL(in, _BOOL);
	IF convertResult THEN
		convertAddress := ADR(_BOOL);
	END_IF
	
	__SYSTEM.TYPE_CLASS.TYPE_BYTE:
	
	convertResult := TryConvert_DINT_TO_BYTE(in, _BYTE);
	IF convertResult THEN
		convertAddress := ADR(_BYTE);
	END_IF
	
	__SYSTEM.TYPE_CLASS.TYPE_WORD:
	
	convertResult := TryConvert_DINT_TO_WORD(in, _WORD);
	IF convertResult THEN
		convertAddress := ADR(_WORD);
	END_IF
	
	__SYSTEM.TYPE_CLASS.TYPE_DWORD:
	
	convertResult := TryConvert_DINT_TO_DWORD(in, _DWORD);
	IF convertResult THEN
		convertAddress := ADR(_DWORD);
	END_IF
	
	__SYSTEM.TYPE_CLASS.TYPE_LWORD:
	
	convertResult := TryConvert_DINT_TO_LWORD(in, _LWORD);
	IF convertResult THEN
		convertAddress := ADR(_LWORD);
	END_IF
	
	__SYSTEM.TYPE_CLASS.TYPE_SINT:
	
	convertResult := TryConvert_DINT_TO_SINT(in, _SINT);
	IF convertResult THEN
		convertAddress := ADR(_SINT);
	END_IF
	
	__SYSTEM.TYPE_CLASS.TYPE_INT:
	
	convertResult := TryConvert_DINT_TO_INT(in, _INT);
	IF convertResult THEN
		convertAddress := ADR(_INT);
	END_IF
	
	__SYSTEM.TYPE_CLASS.TYPE_DINT:
	
	convertResult := TryConvert_DINT_TO_DINT(in, _DINT);
	IF convertResult THEN
		convertAddress := ADR(_DINT);
	END_IF
	
	__SYSTEM.TYPE_CLASS.TYPE_LINT:
	
	convertResult := TryConvert_DINT_TO_LINT(in, _LINT);
	IF convertResult THEN
		convertAddress := ADR(_LINT);
	END_IF
	
	__SYSTEM.TYPE_CLASS.TYPE_USINT:
	
	convertResult := TryConvert_DINT_TO_USINT(in, _USINT);
	IF convertResult THEN
		convertAddress := ADR(_USINT);
	END_IF
	
	__SYSTEM.TYPE_CLASS.TYPE_UINT:
	
	convertResult := TryConvert_DINT_TO_UINT(in, _UINT);
	IF convertResult THEN
		convertAddress := ADR(_UINT);
	END_IF
	
	__SYSTEM.TYPE_CLASS.TYPE_UDINT:
	
	convertResult := TryConvert_DINT_TO_UDINT(in, _UDINT);
	IF convertResult THEN
		convertAddress := ADR(_UDINT);
	END_IF
	
	__SYSTEM.TYPE_CLASS.TYPE_ULINT:
	
	convertResult := TryConvert_DINT_TO_ULINT(in, _ULINT);
	IF convertResult THEN
		convertAddress := ADR(_ULINT);
	END_IF
	
	__SYSTEM.TYPE_CLASS.TYPE_REAL:
	
	convertResult := TryConvert_DINT_TO_REAL(in, _REAL);
	IF convertResult THEN
		convertAddress := ADR(_REAL);
	END_IF
	
	__SYSTEM.TYPE_CLASS.TYPE_LREAL:
	
	convertResult := TryConvert_DINT_TO_LREAL(in, _LREAL);
	IF convertResult THEN
		convertAddress := ADR(_LREAL);
	END_IF
	
	__SYSTEM.TYPE_CLASS.TYPE_TIME:
	
	convertResult := TryConvert_DINT_TO_TIME(in, _TIME);
	IF convertResult THEN
		convertAddress := ADR(_TIME);
	END_IF
	
	__SYSTEM.TYPE_CLASS.TYPE_TIMEOFDAY:
	
	convertResult := TryConvert_DINT_TO_TOD(in, _TOD);
	IF convertResult THEN
		convertAddress := ADR(_TOD);
	END_IF
	
	__SYSTEM.TYPE_CLASS.TYPE_DATE:
	
	convertResult := TryConvert_DINT_TO_DATE(in, _DATE);
	IF convertResult THEN
		convertAddress := ADR(_DATE);
	END_IF
	
	__SYSTEM.TYPE_CLASS.TYPE_DATEANDTIME:
	
	convertResult := TryConvert_DINT_TO_DT(in, _DT);
	IF convertResult THEN
		convertAddress := ADR(_DT);
	END_IF
	
	__SYSTEM.TYPE_CLASS.TYPE_STRING:
	
	convertResult := TryConvert_DINT_TO_STRING(in, _STRING);
	IF convertResult THEN
		convertAddress := ADR(_STRING);
	END_IF
	
END_CASE

IF convertResult THEN
	memcpy(out.pValue,convertAddress,DINT_TO_UDINT(out.diSize));
END_IF

TryConvert_DINT_TO_Destination := convertResult;

END_FUNCTION

// mobject-converters/Converters/DINT_TO_/TryConvert_DINT_TO_WORD
FUNCTION TryConvert_DINT_TO_WORD : BOOL
VAR_INPUT
	in : DINT;
	out : REFERENCE TO WORD;
END_VAR

IF in > DatatypeLimits.MAX_VALUE_OF_DINT_WHICH_CAN_BE_HELD_IN_A_WORD THEN
	RETURN;
END_IF

IF in < DatatypeLimits.MIN_VALUE_OF_DINT_WHICH_CAN_BE_HELD_IN_A_WORD THEN
	RETURN;
END_IF

out := DINT_TO_WORD(in);
TryConvert_DINT_TO_WORD := TRUE;

END_FUNCTION

// mobject-converters/Converters/DINT_TO_/TryConvert_DINT_TO_DWORD
FUNCTION TryConvert_DINT_TO_DWORD : BOOL
VAR_INPUT
	in : DINT;
	out : REFERENCE TO DWORD;
END_VAR

IF in < DatatypeLimits.MIN_VALUE_OF_DINT_WHICH_CAN_BE_HELD_IN_A_DWORD THEN
	RETURN;
END_IF

out := DINT_TO_DWORD(in);
TryConvert_DINT_TO_DWORD := TRUE;

END_FUNCTION

// mobject-converters/Converters/DINT_TO_/TryConvert_DINT_TO_LWORD
FUNCTION TryConvert_DINT_TO_LWORD : BOOL
VAR_INPUT
	in : DINT;
	out : REFERENCE TO LWORD;
END_VAR

IF in < DatatypeLimits.MIN_VALUE_OF_DINT_WHICH_CAN_BE_HELD_IN_A_LWORD THEN
	RETURN;
END_IF

out := DINT_TO_LWORD(in);
TryConvert_DINT_TO_LWORD := TRUE;

END_FUNCTION

// mobject-converters/Converters/DINT_TO_/TryConvert_DINT_TO_SINT
FUNCTION TryConvert_DINT_TO_SINT : BOOL
VAR_INPUT
	in : DINT;
	out : REFERENCE TO SINT;
END_VAR

IF in > DatatypeLimits.MAX_VALUE_OF_DINT_WHICH_CAN_BE_HELD_IN_A_SINT THEN
	RETURN;
END_IF

IF in < DatatypeLimits.MIN_VALUE_OF_DINT_WHICH_CAN_BE_HELD_IN_A_SINT THEN
	RETURN;
END_IF

out := DINT_TO_SINT(in);
TryConvert_DINT_TO_SINT := TRUE;

END_FUNCTION

// mobject-converters/Converters/DINT_TO_/TryConvert_DINT_TO_INT
FUNCTION TryConvert_DINT_TO_INT : BOOL
VAR_INPUT
	in : DINT;
	out : REFERENCE TO INT;
END_VAR

IF in > DatatypeLimits.MAX_VALUE_OF_DINT_WHICH_CAN_BE_HELD_IN_A_INT THEN
	RETURN;
END_IF

IF in < DatatypeLimits.MIN_VALUE_OF_DINT_WHICH_CAN_BE_HELD_IN_A_INT THEN
	RETURN;
END_IF

out := DINT_TO_INT(in);
TryConvert_DINT_TO_INT := TRUE;

END_FUNCTION

// mobject-converters/Converters/DINT_TO_/TryConvert_DINT_TO_DINT
FUNCTION TryConvert_DINT_TO_DINT : BOOL
VAR_INPUT
	in : DINT;
	out : REFERENCE TO DINT;
END_VAR

out := in;
TryConvert_DINT_TO_DINT := TRUE;

END_FUNCTION

// mobject-converters/Converters/DINT_TO_/TryConvert_DINT_TO_LINT
FUNCTION TryConvert_DINT_TO_LINT : BOOL
VAR_INPUT
	in : DINT;
	out : REFERENCE TO LINT;
END_VAR

out := DINT_TO_LINT(in);
TryConvert_DINT_TO_LINT := TRUE;

END_FUNCTION

// mobject-converters/Converters/DINT_TO_/TryConvert_DINT_TO_USINT
FUNCTION TryConvert_DINT_TO_USINT : BOOL
VAR_INPUT
	in : DINT;
	out : REFERENCE TO USINT;
END_VAR

IF in > DatatypeLimits.MAX_VALUE_OF_DINT_WHICH_CAN_BE_HELD_IN_A_USINT THEN
	RETURN;
END_IF

IF in < DatatypeLimits.MIN_VALUE_OF_DINT_WHICH_CAN_BE_HELD_IN_A_USINT THEN
	RETURN;
END_IF

out := DINT_TO_USINT(in);
TryConvert_DINT_TO_USINT := TRUE;

END_FUNCTION

// mobject-converters/Converters/DINT_TO_/TryConvert_DINT_TO_UINT
FUNCTION TryConvert_DINT_TO_UINT : BOOL
VAR_INPUT
	in : DINT;
	out : REFERENCE TO UINT;
END_VAR

IF in > DatatypeLimits.MAX_VALUE_OF_DINT_WHICH_CAN_BE_HELD_IN_A_UINT THEN
	RETURN;
END_IF

IF in < DatatypeLimits.MIN_VALUE_OF_DINT_WHICH_CAN_BE_HELD_IN_A_UINT THEN
	RETURN;
END_IF

out := DINT_TO_UINT(in);
TryConvert_DINT_TO_UINT := TRUE;

END_FUNCTION

// mobject-converters/Converters/DINT_TO_/TryConvert_DINT_TO_UDINT
FUNCTION TryConvert_DINT_TO_UDINT : BOOL
VAR_INPUT
	in : DINT;
	out : REFERENCE TO UDINT;
END_VAR

IF in < DatatypeLimits.MIN_VALUE_OF_DINT_WHICH_CAN_BE_HELD_IN_A_UDINT THEN
	RETURN;
END_IF

out := DINT_TO_UDINT(in);
TryConvert_DINT_TO_UDINT := TRUE;

END_FUNCTION

// mobject-converters/Converters/DINT_TO_/TryConvert_DINT_TO_ULINT
FUNCTION TryConvert_DINT_TO_ULINT : BOOL
VAR_INPUT
	in : DINT;
	out : REFERENCE TO ULINT;
END_VAR

IF in < DatatypeLimits.MIN_VALUE_OF_DINT_WHICH_CAN_BE_HELD_IN_A_ULINT THEN
	RETURN;
END_IF

out := DINT_TO_ULINT(in);
TryConvert_DINT_TO_ULINT := TRUE;

END_FUNCTION

// mobject-converters/Converters/DINT_TO_/TryConvert_DINT_TO_REAL
FUNCTION TryConvert_DINT_TO_REAL : BOOL
VAR_INPUT
	in : DINT;
	out : REFERENCE TO REAL;
END_VAR

out := DINT_TO_REAL(in);
TryConvert_DINT_TO_REAL := TRUE;

END_FUNCTION

// mobject-converters/Converters/DINT_TO_/TryConvert_DINT_TO_LREAL
FUNCTION TryConvert_DINT_TO_LREAL : BOOL
VAR_INPUT
	in : DINT;
	out : REFERENCE TO LREAL;
END_VAR

out := DINT_TO_LREAL(in);
TryConvert_DINT_TO_LREAL := TRUE;

END_FUNCTION

// mobject-converters/Converters/DINT_TO_/TryConvert_DINT_TO_TIME
FUNCTION TryConvert_DINT_TO_TIME : BOOL
VAR_INPUT
	in : DINT;
	out : REFERENCE TO TIME;
END_VAR

IF in < DatatypeLimits.MIN_VALUE_OF_DINT_WHICH_CAN_BE_HELD_IN_A_TIME THEN
	RETURN;
END_IF

out := DINT_TO_TIME(in);
TryConvert_DINT_TO_TIME := TRUE;

END_FUNCTION

// mobject-converters/Converters/DINT_TO_/TryConvert_DINT_TO_TOD
FUNCTION TryConvert_DINT_TO_TOD : BOOL
VAR_INPUT
	in : DINT;
	out : REFERENCE TO TOD;
END_VAR

IF in > DatatypeLimits.MAX_VALUE_OF_DINT_WHICH_CAN_BE_HELD_IN_A_TOD THEN
	RETURN;
END_IF

IF in < DatatypeLimits.MIN_VALUE_OF_DINT_WHICH_CAN_BE_HELD_IN_A_TOD THEN
	RETURN;
END_IF

out := DINT_TO_TOD(in);
TryConvert_DINT_TO_TOD := TRUE;

END_FUNCTION

// mobject-converters/Converters/DINT_TO_/TryConvert_DINT_TO_DT
FUNCTION TryConvert_DINT_TO_DT : BOOL
VAR_INPUT
	in : DINT;
	out : REFERENCE TO DT;
END_VAR

IF in < DatatypeLimits.MIN_VALUE_OF_DINT_WHICH_CAN_BE_HELD_IN_A_DT THEN
	RETURN;
END_IF

out := DINT_TO_DT(in);
TryConvert_DINT_TO_DT := TRUE;

END_FUNCTION

// mobject-converters/Converters/DINT_TO_/TryConvert_DINT_TO_STRING
FUNCTION TryConvert_DINT_TO_STRING : BOOL
VAR_INPUT
	in : DINT;
	out : REFERENCE TO STRING;
END_VAR

out := DINT_TO_STRING(in);
TryConvert_DINT_TO_STRING := TRUE;

END_FUNCTION

// mobject-converters/Converters/DT_TO_/TryConvert_DT_TO_BOOL
FUNCTION TryConvert_DT_TO_BOOL : BOOL
VAR_INPUT
	in : DT;
	out : REFERENCE TO BOOL;
END_VAR

out := DT_TO_BOOL(in);
TryConvert_DT_TO_BOOL := TRUE;

END_FUNCTION

// mobject-converters/Converters/DT_TO_/TryConvert_DT_TO_BYTE
FUNCTION TryConvert_DT_TO_BYTE : BOOL
VAR_INPUT
	in : DT;
	out : REFERENCE TO BYTE;
END_VAR

IF in > DatatypeLimits.MAX_VALUE_OF_DT_WHICH_CAN_BE_HELD_IN_A_BYTE THEN
	RETURN;
END_IF

out := DT_TO_BYTE(in);
TryConvert_DT_TO_BYTE := TRUE;

END_FUNCTION

// mobject-converters/Converters/DT_TO_/TryConvert_DT_TO_DATE
FUNCTION TryConvert_DT_TO_DATE : BOOL
VAR_INPUT
	in : DT;
	out : REFERENCE TO DATE;
END_VAR

out := DT_TO_DATE(in);
TryConvert_DT_TO_DATE := TRUE;

END_FUNCTION

// mobject-converters/Converters/DT_TO_/TryConvert_DT_TO_Destination
FUNCTION TryConvert_DT_TO_Destination : BOOL
VAR_INPUT
	in : DT;
	out : ANY;
END_VAR
VAR
	convertResult : BOOL := FALSE;
	convertAddress : PVOID;
	_BOOL : BOOL;
	_BYTE : BYTE;
	_WORD : WORD;
	_DWORD : DWORD;
	_LWORD : LWORD;
	_SINT : SINT;
	_INT : INT;
	_DINT : DINT;
	_LINT : LINT;
	_USINT : USINT;
	_UINT : UINT;
	_UDINT : UDINT;
	_ULINT : ULINT;
	_REAL : REAL;
	_LREAL : LREAL;
	_TIME : TIME;
	_TOD : TOD;
	_DATE : DATE;
	_DT : DT;
	_STRING : STRING;
END_VAR

CASE out.TypeClass OF
	__SYSTEM.TYPE_CLASS.TYPE_BOOL:
	
	convertResult := TryConvert_DT_TO_BOOL(in, _BOOL);
	IF convertResult THEN
		convertAddress := ADR(_BOOL);
	END_IF
	
	__SYSTEM.TYPE_CLASS.TYPE_BYTE:
	
	convertResult := TryConvert_DT_TO_BYTE(in, _BYTE);
	IF convertResult THEN
		convertAddress := ADR(_BYTE);
	END_IF
	
	__SYSTEM.TYPE_CLASS.TYPE_WORD:
	
	convertResult := TryConvert_DT_TO_WORD(in, _WORD);
	IF convertResult THEN
		convertAddress := ADR(_WORD);
	END_IF
	
	__SYSTEM.TYPE_CLASS.TYPE_DWORD:
	
	convertResult := TryConvert_DT_TO_DWORD(in, _DWORD);
	IF convertResult THEN
		convertAddress := ADR(_DWORD);
	END_IF
	
	__SYSTEM.TYPE_CLASS.TYPE_LWORD:
	
	convertResult := TryConvert_DT_TO_LWORD(in, _LWORD);
	IF convertResult THEN
		convertAddress := ADR(_LWORD);
	END_IF
	
	__SYSTEM.TYPE_CLASS.TYPE_SINT:
	
	convertResult := TryConvert_DT_TO_SINT(in, _SINT);
	IF convertResult THEN
		convertAddress := ADR(_SINT);
	END_IF
	
	__SYSTEM.TYPE_CLASS.TYPE_INT:
	
	convertResult := TryConvert_DT_TO_INT(in, _INT);
	IF convertResult THEN
		convertAddress := ADR(_INT);
	END_IF
	
	__SYSTEM.TYPE_CLASS.TYPE_DINT:
	
	convertResult := TryConvert_DT_TO_DINT(in, _DINT);
	IF convertResult THEN
		convertAddress := ADR(_DINT);
	END_IF
	
	__SYSTEM.TYPE_CLASS.TYPE_LINT:
	
	convertResult := TryConvert_DT_TO_LINT(in, _LINT);
	IF convertResult THEN
		convertAddress := ADR(_LINT);
	END_IF
	
	__SYSTEM.TYPE_CLASS.TYPE_USINT:
	
	convertResult := TryConvert_DT_TO_USINT(in, _USINT);
	IF convertResult THEN
		convertAddress := ADR(_USINT);
	END_IF
	
	__SYSTEM.TYPE_CLASS.TYPE_UINT:
	
	convertResult := TryConvert_DT_TO_UINT(in, _UINT);
	IF convertResult THEN
		convertAddress := ADR(_UINT);
	END_IF
	
	__SYSTEM.TYPE_CLASS.TYPE_UDINT:
	
	convertResult := TryConvert_DT_TO_UDINT(in, _UDINT);
	IF convertResult THEN
		convertAddress := ADR(_UDINT);
	END_IF
	
	__SYSTEM.TYPE_CLASS.TYPE_ULINT:
	
	convertResult := TryConvert_DT_TO_ULINT(in, _ULINT);
	IF convertResult THEN
		convertAddress := ADR(_ULINT);
	END_IF
	
	__SYSTEM.TYPE_CLASS.TYPE_REAL:
	
	convertResult := TryConvert_DT_TO_REAL(in, _REAL);
	IF convertResult THEN
		convertAddress := ADR(_REAL);
	END_IF
	
	__SYSTEM.TYPE_CLASS.TYPE_LREAL:
	
	convertResult := TryConvert_DT_TO_LREAL(in, _LREAL);
	IF convertResult THEN
		convertAddress := ADR(_LREAL);
	END_IF
	
	__SYSTEM.TYPE_CLASS.TYPE_TIME:
	
	convertResult := TryConvert_DT_TO_TIME(in, _TIME);
	IF convertResult THEN
		convertAddress := ADR(_TIME);
	END_IF
	
	__SYSTEM.TYPE_CLASS.TYPE_TIMEOFDAY:
	
	convertResult := TryConvert_DT_TO_TOD(in, _TOD);
	IF convertResult THEN
		convertAddress := ADR(_TOD);
	END_IF
	
	__SYSTEM.TYPE_CLASS.TYPE_DATE:
	
	convertResult := TryConvert_DT_TO_DATE(in, _DATE);
	IF convertResult THEN
		convertAddress := ADR(_DATE);
	END_IF
	
	__SYSTEM.TYPE_CLASS.TYPE_DATEANDTIME:
	
	convertResult := TryConvert_DT_TO_DT(in, _DT);
	IF convertResult THEN
		convertAddress := ADR(_DT);
	END_IF
	
	__SYSTEM.TYPE_CLASS.TYPE_STRING:
	
	convertResult := TryConvert_DT_TO_STRING(in, _STRING);
	IF convertResult THEN
		convertAddress := ADR(_STRING);
	END_IF
	
END_CASE

IF convertResult THEN
	memcpy(out.pValue,convertAddress,DINT_TO_UDINT(out.diSize));
END_IF

TryConvert_DT_TO_Destination := convertResult;

END_FUNCTION

// mobject-converters/Converters/DT_TO_/TryConvert_DT_TO_WORD
FUNCTION TryConvert_DT_TO_WORD : BOOL
VAR_INPUT
	in : DT;
	out : REFERENCE TO WORD;
END_VAR

IF in > DatatypeLimits.MAX_VALUE_OF_DT_WHICH_CAN_BE_HELD_IN_A_WORD THEN
	RETURN;
END_IF

out := DT_TO_WORD(in);
TryConvert_DT_TO_WORD := TRUE;

END_FUNCTION

// mobject-converters/Converters/DT_TO_/TryConvert_DT_TO_DWORD
FUNCTION TryConvert_DT_TO_DWORD : BOOL
VAR_INPUT
	in : DT;
	out : REFERENCE TO DWORD;
END_VAR

out := DT_TO_DWORD(in);
TryConvert_DT_TO_DWORD := TRUE;

END_FUNCTION

// mobject-converters/Converters/DT_TO_/TryConvert_DT_TO_LWORD
FUNCTION TryConvert_DT_TO_LWORD : BOOL
VAR_INPUT
	in : DT;
	out : REFERENCE TO LWORD;
END_VAR

out := DT_TO_LWORD(in);
TryConvert_DT_TO_LWORD := TRUE;

END_FUNCTION

// mobject-converters/Converters/DT_TO_/TryConvert_DT_TO_SINT
FUNCTION TryConvert_DT_TO_SINT : BOOL
VAR_INPUT
	in : DT;
	out : REFERENCE TO SINT;
END_VAR

IF in > DatatypeLimits.MAX_VALUE_OF_DT_WHICH_CAN_BE_HELD_IN_A_SINT THEN
	RETURN;
END_IF

out := DT_TO_SINT(in);
TryConvert_DT_TO_SINT := TRUE;

END_FUNCTION

// mobject-converters/Converters/DT_TO_/TryConvert_DT_TO_INT
FUNCTION TryConvert_DT_TO_INT : BOOL
VAR_INPUT
	in : DT;
	out : REFERENCE TO INT;
END_VAR

IF in > DatatypeLimits.MAX_VALUE_OF_DT_WHICH_CAN_BE_HELD_IN_A_INT THEN
	RETURN;
END_IF

out := DT_TO_INT(in);
TryConvert_DT_TO_INT := TRUE;

END_FUNCTION

// mobject-converters/Converters/DT_TO_/TryConvert_DT_TO_DINT
FUNCTION TryConvert_DT_TO_DINT : BOOL
VAR_INPUT
	in : DT;
	out : REFERENCE TO DINT;
END_VAR

IF in > DatatypeLimits.MAX_VALUE_OF_DT_WHICH_CAN_BE_HELD_IN_A_DINT THEN
	RETURN;
END_IF

out := DT_TO_DINT(in);
TryConvert_DT_TO_DINT := TRUE;

END_FUNCTION

// mobject-converters/Converters/DT_TO_/TryConvert_DT_TO_LINT
FUNCTION TryConvert_DT_TO_LINT : BOOL
VAR_INPUT
	in : DT;
	out : REFERENCE TO LINT;
END_VAR

out := DT_TO_LINT(in);
TryConvert_DT_TO_LINT := TRUE;

END_FUNCTION

// mobject-converters/Converters/DT_TO_/TryConvert_DT_TO_USINT
FUNCTION TryConvert_DT_TO_USINT : BOOL
VAR_INPUT
	in : DT;
	out : REFERENCE TO USINT;
END_VAR

IF in > DatatypeLimits.MAX_VALUE_OF_DT_WHICH_CAN_BE_HELD_IN_A_USINT THEN
	RETURN;
END_IF

out := DT_TO_USINT(in);
TryConvert_DT_TO_USINT := TRUE;

END_FUNCTION

// mobject-converters/Converters/DT_TO_/TryConvert_DT_TO_UINT
FUNCTION TryConvert_DT_TO_UINT : BOOL
VAR_INPUT
	in : DT;
	out : REFERENCE TO UINT;
END_VAR

IF in > DatatypeLimits.MAX_VALUE_OF_DT_WHICH_CAN_BE_HELD_IN_A_UINT THEN
	RETURN;
END_IF

out := DT_TO_UINT(in);
TryConvert_DT_TO_UINT := TRUE;

END_FUNCTION

// mobject-converters/Converters/DT_TO_/TryConvert_DT_TO_UDINT
FUNCTION TryConvert_DT_TO_UDINT : BOOL
VAR_INPUT
	in : DT;
	out : REFERENCE TO UDINT;
END_VAR

out := DT_TO_UDINT(in);
TryConvert_DT_TO_UDINT := TRUE;

END_FUNCTION

// mobject-converters/Converters/DT_TO_/TryConvert_DT_TO_ULINT
FUNCTION TryConvert_DT_TO_ULINT : BOOL
VAR_INPUT
	in : DT;
	out : REFERENCE TO ULINT;
END_VAR

out := DT_TO_ULINT(in);
TryConvert_DT_TO_ULINT := TRUE;

END_FUNCTION

// mobject-converters/Converters/DT_TO_/TryConvert_DT_TO_REAL
FUNCTION TryConvert_DT_TO_REAL : BOOL
VAR_INPUT
	in : DT;
	out : REFERENCE TO REAL;
END_VAR

out := DT_TO_REAL(in);
TryConvert_DT_TO_REAL := TRUE;

END_FUNCTION

// mobject-converters/Converters/DT_TO_/TryConvert_DT_TO_LREAL
FUNCTION TryConvert_DT_TO_LREAL : BOOL
VAR_INPUT
	in : DT;
	out : REFERENCE TO LREAL;
END_VAR

out := DT_TO_LREAL(in);
TryConvert_DT_TO_LREAL := TRUE;

END_FUNCTION

// mobject-converters/Converters/DT_TO_/TryConvert_DT_TO_TIME
FUNCTION TryConvert_DT_TO_TIME : BOOL
VAR_INPUT
	in : DT;
	out : REFERENCE TO TIME;
END_VAR

IF in > DatatypeLimits.MAX_VALUE_OF_DT_WHICH_CAN_BE_HELD_IN_A_TIME THEN
	RETURN;
END_IF

out := DT_TO_TIME(in);
TryConvert_DT_TO_TIME := TRUE;

END_FUNCTION

// mobject-converters/Converters/DT_TO_/TryConvert_DT_TO_TOD
FUNCTION TryConvert_DT_TO_TOD : BOOL
VAR_INPUT
	in : DT;
	out : REFERENCE TO TOD;
END_VAR

IF in > DatatypeLimits.MAX_VALUE_OF_DT_WHICH_CAN_BE_HELD_IN_A_TOD THEN
	RETURN;
END_IF

out := DT_TO_TOD(in);
TryConvert_DT_TO_TOD := TRUE;

END_FUNCTION

// mobject-converters/Converters/DT_TO_/TryConvert_DT_TO_DT
FUNCTION TryConvert_DT_TO_DT : BOOL
VAR_INPUT
	in : DT;
	out : REFERENCE TO DT;
END_VAR

out := in;
TryConvert_DT_TO_DT := TRUE;

END_FUNCTION

// mobject-converters/Converters/DT_TO_/TryConvert_DT_TO_STRING
FUNCTION TryConvert_DT_TO_STRING : BOOL
VAR_INPUT
	in : DT;
	out : REFERENCE TO STRING;
END_VAR

out := DT_TO_STRING(in);
TryConvert_DT_TO_STRING := TRUE;

END_FUNCTION

// mobject-converters/Converters/DWORD_TO_/TryConvert_DWORD_TO_BOOL
FUNCTION TryConvert_DWORD_TO_BOOL : BOOL
VAR_INPUT
	in : DWORD;
	out : REFERENCE TO BOOL;
END_VAR

out := DWORD_TO_BOOL(in);
TryConvert_DWORD_TO_BOOL := TRUE;

END_FUNCTION

// mobject-converters/Converters/DWORD_TO_/TryConvert_DWORD_TO_BYTE
FUNCTION TryConvert_DWORD_TO_BYTE : BOOL
VAR_INPUT
	in : DWORD;
	out : REFERENCE TO BYTE;
END_VAR

IF in > DatatypeLimits.MAX_VALUE_OF_DWORD_WHICH_CAN_BE_HELD_IN_A_BYTE THEN
	RETURN;
END_IF

out := DWORD_TO_BYTE(in);
TryConvert_DWORD_TO_BYTE := TRUE;

END_FUNCTION

// mobject-converters/Converters/DWORD_TO_/TryConvert_DWORD_TO_DATE
FUNCTION TryConvert_DWORD_TO_DATE : BOOL
VAR_INPUT
	in : DWORD;
	out : REFERENCE TO DATE;
END_VAR

out := DWORD_TO_DATE(in);
TryConvert_DWORD_TO_DATE := TRUE;

END_FUNCTION

// mobject-converters/Converters/DWORD_TO_/TryConvert_DWORD_TO_Destination
FUNCTION TryConvert_DWORD_TO_Destination : BOOL
VAR_INPUT
	in : DWORD;
	out : ANY;
END_VAR
VAR
	convertResult : BOOL := FALSE;
	convertAddress : PVOID;
	_BOOL : BOOL;
	_BYTE : BYTE;
	_WORD : WORD;
	_DWORD : DWORD;
	_LWORD : LWORD;
	_SINT : SINT;
	_INT : INT;
	_DINT : DINT;
	_LINT : LINT;
	_USINT : USINT;
	_UINT : UINT;
	_UDINT : UDINT;
	_ULINT : ULINT;
	_REAL : REAL;
	_LREAL : LREAL;
	_TIME : TIME;
	_TOD : TOD;
	_DATE : DATE;
	_DT : DT;
	_STRING : STRING;
END_VAR

CASE out.TypeClass OF
	__SYSTEM.TYPE_CLASS.TYPE_BOOL:
	
	convertResult := TryConvert_DWORD_TO_BOOL(in, _BOOL);
	IF convertResult THEN
		convertAddress := ADR(_BOOL);
	END_IF
	
	__SYSTEM.TYPE_CLASS.TYPE_BYTE:
	
	convertResult := TryConvert_DWORD_TO_BYTE(in, _BYTE);
	IF convertResult THEN
		convertAddress := ADR(_BYTE);
	END_IF
	
	__SYSTEM.TYPE_CLASS.TYPE_WORD:
	
	convertResult := TryConvert_DWORD_TO_WORD(in, _WORD);
	IF convertResult THEN
		convertAddress := ADR(_WORD);
	END_IF
	
	__SYSTEM.TYPE_CLASS.TYPE_DWORD:
	
	convertResult := TryConvert_DWORD_TO_DWORD(in, _DWORD);
	IF convertResult THEN
		convertAddress := ADR(_DWORD);
	END_IF
	
	__SYSTEM.TYPE_CLASS.TYPE_LWORD:
	
	convertResult := TryConvert_DWORD_TO_LWORD(in, _LWORD);
	IF convertResult THEN
		convertAddress := ADR(_LWORD);
	END_IF
	
	__SYSTEM.TYPE_CLASS.TYPE_SINT:
	
	convertResult := TryConvert_DWORD_TO_SINT(in, _SINT);
	IF convertResult THEN
		convertAddress := ADR(_SINT);
	END_IF
	
	__SYSTEM.TYPE_CLASS.TYPE_INT:
	
	convertResult := TryConvert_DWORD_TO_INT(in, _INT);
	IF convertResult THEN
		convertAddress := ADR(_INT);
	END_IF
	
	__SYSTEM.TYPE_CLASS.TYPE_DINT:
	
	convertResult := TryConvert_DWORD_TO_DINT(in, _DINT);
	IF convertResult THEN
		convertAddress := ADR(_DINT);
	END_IF
	
	__SYSTEM.TYPE_CLASS.TYPE_LINT:
	
	convertResult := TryConvert_DWORD_TO_LINT(in, _LINT);
	IF convertResult THEN
		convertAddress := ADR(_LINT);
	END_IF
	
	__SYSTEM.TYPE_CLASS.TYPE_USINT:
	
	convertResult := TryConvert_DWORD_TO_USINT(in, _USINT);
	IF convertResult THEN
		convertAddress := ADR(_USINT);
	END_IF
	
	__SYSTEM.TYPE_CLASS.TYPE_UINT:
	
	convertResult := TryConvert_DWORD_TO_UINT(in, _UINT);
	IF convertResult THEN
		convertAddress := ADR(_UINT);
	END_IF
	
	__SYSTEM.TYPE_CLASS.TYPE_UDINT:
	
	convertResult := TryConvert_DWORD_TO_UDINT(in, _UDINT);
	IF convertResult THEN
		convertAddress := ADR(_UDINT);
	END_IF
	
	__SYSTEM.TYPE_CLASS.TYPE_ULINT:
	
	convertResult := TryConvert_DWORD_TO_ULINT(in, _ULINT);
	IF convertResult THEN
		convertAddress := ADR(_ULINT);
	END_IF
	
	__SYSTEM.TYPE_CLASS.TYPE_REAL:
	
	convertResult := TryConvert_DWORD_TO_REAL(in, _REAL);
	IF convertResult THEN
		convertAddress := ADR(_REAL);
	END_IF
	
	__SYSTEM.TYPE_CLASS.TYPE_LREAL:
	
	convertResult := TryConvert_DWORD_TO_LREAL(in, _LREAL);
	IF convertResult THEN
		convertAddress := ADR(_LREAL);
	END_IF
	
	__SYSTEM.TYPE_CLASS.TYPE_TIME:
	
	convertResult := TryConvert_DWORD_TO_TIME(in, _TIME);
	IF convertResult THEN
		convertAddress := ADR(_TIME);
	END_IF
	
	__SYSTEM.TYPE_CLASS.TYPE_TIMEOFDAY:
	
	convertResult := TryConvert_DWORD_TO_TOD(in, _TOD);
	IF convertResult THEN
		convertAddress := ADR(_TOD);
	END_IF
	
	__SYSTEM.TYPE_CLASS.TYPE_DATE:
	
	convertResult := TryConvert_DWORD_TO_DATE(in, _DATE);
	IF convertResult THEN
		convertAddress := ADR(_DATE);
	END_IF
	
	__SYSTEM.TYPE_CLASS.TYPE_DATEANDTIME:
	
	convertResult := TryConvert_DWORD_TO_DT(in, _DT);
	IF convertResult THEN
		convertAddress := ADR(_DT);
	END_IF
	
	__SYSTEM.TYPE_CLASS.TYPE_STRING:
	
	convertResult := TryConvert_DWORD_TO_STRING(in, _STRING);
	IF convertResult THEN
		convertAddress := ADR(_STRING);
	END_IF
	
END_CASE

IF convertResult THEN
	memcpy(out.pValue,convertAddress,DINT_TO_UDINT(out.diSize));
END_IF

TryConvert_DWORD_TO_Destination := convertResult;

END_FUNCTION

// mobject-converters/Converters/DWORD_TO_/TryConvert_DWORD_TO_WORD
FUNCTION TryConvert_DWORD_TO_WORD : BOOL
VAR_INPUT
	in : DWORD;
	out : REFERENCE TO WORD;
END_VAR

IF in > DatatypeLimits.MAX_VALUE_OF_DWORD_WHICH_CAN_BE_HELD_IN_A_WORD THEN
	RETURN;
END_IF

out := DWORD_TO_WORD(in);
TryConvert_DWORD_TO_WORD := TRUE;

END_FUNCTION

// mobject-converters/Converters/DWORD_TO_/TryConvert_DWORD_TO_DWORD
FUNCTION TryConvert_DWORD_TO_DWORD : BOOL
VAR_INPUT
	in : DWORD;
	out : REFERENCE TO DWORD;
END_VAR

out := in;
TryConvert_DWORD_TO_DWORD := TRUE;

END_FUNCTION

// mobject-converters/Converters/DWORD_TO_/TryConvert_DWORD_TO_LWORD
FUNCTION TryConvert_DWORD_TO_LWORD : BOOL
VAR_INPUT
	in : DWORD;
	out : REFERENCE TO LWORD;
END_VAR

out := DWORD_TO_LWORD(in);
TryConvert_DWORD_TO_LWORD := TRUE;

END_FUNCTION

// mobject-converters/Converters/DWORD_TO_/TryConvert_DWORD_TO_SINT
FUNCTION TryConvert_DWORD_TO_SINT : BOOL
VAR_INPUT
	in : DWORD;
	out : REFERENCE TO SINT;
END_VAR

IF in > DatatypeLimits.MAX_VALUE_OF_DWORD_WHICH_CAN_BE_HELD_IN_A_SINT THEN
	RETURN;
END_IF

out := DWORD_TO_SINT(in);
TryConvert_DWORD_TO_SINT := TRUE;

END_FUNCTION

// mobject-converters/Converters/DWORD_TO_/TryConvert_DWORD_TO_INT
FUNCTION TryConvert_DWORD_TO_INT : BOOL
VAR_INPUT
	in : DWORD;
	out : REFERENCE TO INT;
END_VAR

IF in > DatatypeLimits.MAX_VALUE_OF_DWORD_WHICH_CAN_BE_HELD_IN_A_INT THEN
	RETURN;
END_IF

out := DWORD_TO_INT(in);
TryConvert_DWORD_TO_INT := TRUE;

END_FUNCTION

// mobject-converters/Converters/DWORD_TO_/TryConvert_DWORD_TO_DINT
FUNCTION TryConvert_DWORD_TO_DINT : BOOL
VAR_INPUT
	in : DWORD;
	out : REFERENCE TO DINT;
END_VAR

IF in > DatatypeLimits.MAX_VALUE_OF_DWORD_WHICH_CAN_BE_HELD_IN_A_DINT THEN
	RETURN;
END_IF

out := DWORD_TO_DINT(in);
TryConvert_DWORD_TO_DINT := TRUE;

END_FUNCTION

// mobject-converters/Converters/DWORD_TO_/TryConvert_DWORD_TO_LINT
FUNCTION TryConvert_DWORD_TO_LINT : BOOL
VAR_INPUT
	in : DWORD;
	out : REFERENCE TO LINT;
END_VAR

out := DWORD_TO_LINT(in);
TryConvert_DWORD_TO_LINT := TRUE;

END_FUNCTION

// mobject-converters/Converters/DWORD_TO_/TryConvert_DWORD_TO_USINT
FUNCTION TryConvert_DWORD_TO_USINT : BOOL
VAR_INPUT
	in : DWORD;
	out : REFERENCE TO USINT;
END_VAR

IF in > DatatypeLimits.MAX_VALUE_OF_DWORD_WHICH_CAN_BE_HELD_IN_A_USINT THEN
	RETURN;
END_IF

out := DWORD_TO_USINT(in);
TryConvert_DWORD_TO_USINT := TRUE;

END_FUNCTION

// mobject-converters/Converters/DWORD_TO_/TryConvert_DWORD_TO_UINT
FUNCTION TryConvert_DWORD_TO_UINT : BOOL
VAR_INPUT
	in : DWORD;
	out : REFERENCE TO UINT;
END_VAR

IF in > DatatypeLimits.MAX_VALUE_OF_DWORD_WHICH_CAN_BE_HELD_IN_A_UINT THEN
	RETURN;
END_IF

out := DWORD_TO_UINT(in);
TryConvert_DWORD_TO_UINT := TRUE;

END_FUNCTION

// mobject-converters/Converters/DWORD_TO_/TryConvert_DWORD_TO_UDINT
FUNCTION TryConvert_DWORD_TO_UDINT : BOOL
VAR_INPUT
	in : DWORD;
	out : REFERENCE TO UDINT;
END_VAR

out := DWORD_TO_UDINT(in);
TryConvert_DWORD_TO_UDINT := TRUE;

END_FUNCTION

// mobject-converters/Converters/DWORD_TO_/TryConvert_DWORD_TO_ULINT
FUNCTION TryConvert_DWORD_TO_ULINT : BOOL
VAR_INPUT
	in : DWORD;
	out : REFERENCE TO ULINT;
END_VAR

out := DWORD_TO_ULINT(in);
TryConvert_DWORD_TO_ULINT := TRUE;

END_FUNCTION

// mobject-converters/Converters/DWORD_TO_/TryConvert_DWORD_TO_REAL
FUNCTION TryConvert_DWORD_TO_REAL : BOOL
VAR_INPUT
	in : DWORD;
	out : REFERENCE TO REAL;
END_VAR

out := DWORD_TO_REAL(in);
TryConvert_DWORD_TO_REAL := TRUE;

END_FUNCTION

// mobject-converters/Converters/DWORD_TO_/TryConvert_DWORD_TO_LREAL
FUNCTION TryConvert_DWORD_TO_LREAL : BOOL
VAR_INPUT
	in : DWORD;
	out : REFERENCE TO LREAL;
END_VAR

out := DWORD_TO_LREAL(in);
TryConvert_DWORD_TO_LREAL := TRUE;

END_FUNCTION

// mobject-converters/Converters/DWORD_TO_/TryConvert_DWORD_TO_TIME
FUNCTION TryConvert_DWORD_TO_TIME : BOOL
VAR_INPUT
	in : DWORD;
	out : REFERENCE TO TIME;
END_VAR

out := DWORD_TO_TIME(in);
TryConvert_DWORD_TO_TIME := TRUE;

END_FUNCTION

// mobject-converters/Converters/DWORD_TO_/TryConvert_DWORD_TO_TOD
FUNCTION TryConvert_DWORD_TO_TOD : BOOL
VAR_INPUT
	in : DWORD;
	out : REFERENCE TO TOD;
END_VAR

IF in > DatatypeLimits.MAX_VALUE_OF_DWORD_WHICH_CAN_BE_HELD_IN_A_TOD THEN
	RETURN;
END_IF

out := DWORD_TO_TOD(in);
TryConvert_DWORD_TO_TOD := TRUE;

END_FUNCTION

// mobject-converters/Converters/DWORD_TO_/TryConvert_DWORD_TO_DT
FUNCTION TryConvert_DWORD_TO_DT : BOOL
VAR_INPUT
	in : DWORD;
	out : REFERENCE TO DT;
END_VAR

out := DWORD_TO_DT(in);
TryConvert_DWORD_TO_DT := TRUE;

END_FUNCTION

// mobject-converters/Converters/DWORD_TO_/TryConvert_DWORD_TO_STRING
FUNCTION TryConvert_DWORD_TO_STRING : BOOL
VAR_INPUT
	in : DWORD;
	out : REFERENCE TO STRING;
END_VAR

out := DWORD_TO_STRING(in);
TryConvert_DWORD_TO_STRING := TRUE;

END_FUNCTION

// mobject-converters/Converters/INT_TO_/TryConvert_INT_TO_BOOL
FUNCTION TryConvert_INT_TO_BOOL : BOOL
VAR_INPUT
	in : INT;
	out : REFERENCE TO BOOL;
END_VAR

out := INT_TO_BOOL(in);
TryConvert_INT_TO_BOOL := TRUE;

END_FUNCTION

// mobject-converters/Converters/INT_TO_/TryConvert_INT_TO_BYTE
FUNCTION TryConvert_INT_TO_BYTE : BOOL
VAR_INPUT
	in : INT;
	out : REFERENCE TO BYTE;
END_VAR

IF in > DatatypeLimits.MAX_VALUE_OF_INT_WHICH_CAN_BE_HELD_IN_A_BYTE THEN
	RETURN;
END_IF

IF in < DatatypeLimits.MIN_VALUE_OF_INT_WHICH_CAN_BE_HELD_IN_A_BYTE THEN
	RETURN;
END_IF

out := INT_TO_BYTE(in);
TryConvert_INT_TO_BYTE := TRUE;

END_FUNCTION

// mobject-converters/Converters/INT_TO_/TryConvert_INT_TO_DATE
FUNCTION TryConvert_INT_TO_DATE : BOOL
VAR_INPUT
	in : INT;
	out : REFERENCE TO DATE;
END_VAR

IF in < DatatypeLimits.MIN_VALUE_OF_INT_WHICH_CAN_BE_HELD_IN_A_DATE THEN
	RETURN;
END_IF

out := INT_TO_DATE(in);
TryConvert_INT_TO_DATE := TRUE;

END_FUNCTION

// mobject-converters/Converters/INT_TO_/TryConvert_INT_TO_Destination
FUNCTION TryConvert_INT_TO_Destination : BOOL
VAR_INPUT
	in : INT;
	out : ANY;
END_VAR
VAR
	convertResult : BOOL := FALSE;
	convertAddress : PVOID;
	_BOOL : BOOL;
	_BYTE : BYTE;
	_WORD : WORD;
	_DWORD : DWORD;
	_LWORD : LWORD;
	_SINT : SINT;
	_INT : INT;
	_DINT : DINT;
	_LINT : LINT;
	_USINT : USINT;
	_UINT : UINT;
	_UDINT : UDINT;
	_ULINT : ULINT;
	_REAL : REAL;
	_LREAL : LREAL;
	_TIME : TIME;
	_TOD : TOD;
	_DATE : DATE;
	_DT : DT;
	_STRING : STRING;
END_VAR

CASE out.TypeClass OF
	__SYSTEM.TYPE_CLASS.TYPE_BOOL:
	
	convertResult := TryConvert_INT_TO_BOOL(in, _BOOL);
	IF convertResult THEN
		convertAddress := ADR(_BOOL);
	END_IF
	
	__SYSTEM.TYPE_CLASS.TYPE_BYTE:
	
	convertResult := TryConvert_INT_TO_BYTE(in, _BYTE);
	IF convertResult THEN
		convertAddress := ADR(_BYTE);
	END_IF
	
	__SYSTEM.TYPE_CLASS.TYPE_WORD:
	
	convertResult := TryConvert_INT_TO_WORD(in, _WORD);
	IF convertResult THEN
		convertAddress := ADR(_WORD);
	END_IF
	
	__SYSTEM.TYPE_CLASS.TYPE_DWORD:
	
	convertResult := TryConvert_INT_TO_DWORD(in, _DWORD);
	IF convertResult THEN
		convertAddress := ADR(_DWORD);
	END_IF
	
	__SYSTEM.TYPE_CLASS.TYPE_LWORD:
	
	convertResult := TryConvert_INT_TO_LWORD(in, _LWORD);
	IF convertResult THEN
		convertAddress := ADR(_LWORD);
	END_IF
	
	__SYSTEM.TYPE_CLASS.TYPE_SINT:
	
	convertResult := TryConvert_INT_TO_SINT(in, _SINT);
	IF convertResult THEN
		convertAddress := ADR(_SINT);
	END_IF
	
	__SYSTEM.TYPE_CLASS.TYPE_INT:
	
	convertResult := TryConvert_INT_TO_INT(in, _INT);
	IF convertResult THEN
		convertAddress := ADR(_INT);
	END_IF
	
	__SYSTEM.TYPE_CLASS.TYPE_DINT:
	
	convertResult := TryConvert_INT_TO_DINT(in, _DINT);
	IF convertResult THEN
		convertAddress := ADR(_DINT);
	END_IF
	
	__SYSTEM.TYPE_CLASS.TYPE_LINT:
	
	convertResult := TryConvert_INT_TO_LINT(in, _LINT);
	IF convertResult THEN
		convertAddress := ADR(_LINT);
	END_IF
	
	__SYSTEM.TYPE_CLASS.TYPE_USINT:
	
	convertResult := TryConvert_INT_TO_USINT(in, _USINT);
	IF convertResult THEN
		convertAddress := ADR(_USINT);
	END_IF
	
	__SYSTEM.TYPE_CLASS.TYPE_UINT:
	
	convertResult := TryConvert_INT_TO_UINT(in, _UINT);
	IF convertResult THEN
		convertAddress := ADR(_UINT);
	END_IF
	
	__SYSTEM.TYPE_CLASS.TYPE_UDINT:
	
	convertResult := TryConvert_INT_TO_UDINT(in, _UDINT);
	IF convertResult THEN
		convertAddress := ADR(_UDINT);
	END_IF
	
	__SYSTEM.TYPE_CLASS.TYPE_ULINT:
	
	convertResult := TryConvert_INT_TO_ULINT(in, _ULINT);
	IF convertResult THEN
		convertAddress := ADR(_ULINT);
	END_IF
	
	__SYSTEM.TYPE_CLASS.TYPE_REAL:
	
	convertResult := TryConvert_INT_TO_REAL(in, _REAL);
	IF convertResult THEN
		convertAddress := ADR(_REAL);
	END_IF
	
	__SYSTEM.TYPE_CLASS.TYPE_LREAL:
	
	convertResult := TryConvert_INT_TO_LREAL(in, _LREAL);
	IF convertResult THEN
		convertAddress := ADR(_LREAL);
	END_IF
	
	__SYSTEM.TYPE_CLASS.TYPE_TIME:
	
	convertResult := TryConvert_INT_TO_TIME(in, _TIME);
	IF convertResult THEN
		convertAddress := ADR(_TIME);
	END_IF
	
	__SYSTEM.TYPE_CLASS.TYPE_TIMEOFDAY:
	
	convertResult := TryConvert_INT_TO_TOD(in, _TOD);
	IF convertResult THEN
		convertAddress := ADR(_TOD);
	END_IF
	
	__SYSTEM.TYPE_CLASS.TYPE_DATE:
	
	convertResult := TryConvert_INT_TO_DATE(in, _DATE);
	IF convertResult THEN
		convertAddress := ADR(_DATE);
	END_IF
	
	__SYSTEM.TYPE_CLASS.TYPE_DATEANDTIME:
	
	convertResult := TryConvert_INT_TO_DT(in, _DT);
	IF convertResult THEN
		convertAddress := ADR(_DT);
	END_IF
	
	__SYSTEM.TYPE_CLASS.TYPE_STRING:
	
	convertResult := TryConvert_INT_TO_STRING(in, _STRING);
	IF convertResult THEN
		convertAddress := ADR(_STRING);
	END_IF
	
END_CASE

IF convertResult THEN
	memcpy(out.pValue,convertAddress,DINT_TO_UDINT(out.diSize));
END_IF

TryConvert_INT_TO_Destination := convertResult;

END_FUNCTION

// mobject-converters/Converters/INT_TO_/TryConvert_INT_TO_WORD
FUNCTION TryConvert_INT_TO_WORD : BOOL
VAR_INPUT
	in : INT;
	out : REFERENCE TO WORD;
END_VAR

IF in < DatatypeLimits.MIN_VALUE_OF_INT_WHICH_CAN_BE_HELD_IN_A_WORD THEN
	RETURN;
END_IF

out := INT_TO_WORD(in);
TryConvert_INT_TO_WORD := TRUE;

END_FUNCTION

// mobject-converters/Converters/INT_TO_/TryConvert_INT_TO_DWORD
FUNCTION TryConvert_INT_TO_DWORD : BOOL
VAR_INPUT
	in : INT;
	out : REFERENCE TO DWORD;
END_VAR

IF in < DatatypeLimits.MIN_VALUE_OF_INT_WHICH_CAN_BE_HELD_IN_A_DWORD THEN
	RETURN;
END_IF

out := INT_TO_DWORD(in);
TryConvert_INT_TO_DWORD := TRUE;

END_FUNCTION

// mobject-converters/Converters/INT_TO_/TryConvert_INT_TO_LWORD
FUNCTION TryConvert_INT_TO_LWORD : BOOL
VAR_INPUT
	in : INT;
	out : REFERENCE TO LWORD;
END_VAR

IF in < DatatypeLimits.MIN_VALUE_OF_INT_WHICH_CAN_BE_HELD_IN_A_LWORD THEN
	RETURN;
END_IF

out := INT_TO_LWORD(in);
TryConvert_INT_TO_LWORD := TRUE;

END_FUNCTION

// mobject-converters/Converters/INT_TO_/TryConvert_INT_TO_SINT
FUNCTION TryConvert_INT_TO_SINT : BOOL
VAR_INPUT
	in : INT;
	out : REFERENCE TO SINT;
END_VAR

IF in > DatatypeLimits.MAX_VALUE_OF_INT_WHICH_CAN_BE_HELD_IN_A_SINT THEN
	RETURN;
END_IF

IF in < DatatypeLimits.MIN_VALUE_OF_INT_WHICH_CAN_BE_HELD_IN_A_SINT THEN
	RETURN;
END_IF

out := INT_TO_SINT(in);
TryConvert_INT_TO_SINT := TRUE;

END_FUNCTION

// mobject-converters/Converters/INT_TO_/TryConvert_INT_TO_INT
FUNCTION TryConvert_INT_TO_INT : BOOL
VAR_INPUT
	in : INT;
	out : REFERENCE TO INT;
END_VAR

out := in;
TryConvert_INT_TO_INT := TRUE;

END_FUNCTION

// mobject-converters/Converters/INT_TO_/TryConvert_INT_TO_DINT
FUNCTION TryConvert_INT_TO_DINT : BOOL
VAR_INPUT
	in : INT;
	out : REFERENCE TO DINT;
END_VAR

out := INT_TO_DINT(in);
TryConvert_INT_TO_DINT := TRUE;

END_FUNCTION

// mobject-converters/Converters/INT_TO_/TryConvert_INT_TO_LINT
FUNCTION TryConvert_INT_TO_LINT : BOOL
VAR_INPUT
	in : INT;
	out : REFERENCE TO LINT;
END_VAR

out := INT_TO_LINT(in);
TryConvert_INT_TO_LINT := TRUE;

END_FUNCTION

// mobject-converters/Converters/INT_TO_/TryConvert_INT_TO_USINT
FUNCTION TryConvert_INT_TO_USINT : BOOL
VAR_INPUT
	in : INT;
	out : REFERENCE TO USINT;
END_VAR

IF in > DatatypeLimits.MAX_VALUE_OF_INT_WHICH_CAN_BE_HELD_IN_A_USINT THEN
	RETURN;
END_IF

IF in < DatatypeLimits.MIN_VALUE_OF_INT_WHICH_CAN_BE_HELD_IN_A_USINT THEN
	RETURN;
END_IF

out := INT_TO_USINT(in);
TryConvert_INT_TO_USINT := TRUE;

END_FUNCTION

// mobject-converters/Converters/INT_TO_/TryConvert_INT_TO_UINT
FUNCTION TryConvert_INT_TO_UINT : BOOL
VAR_INPUT
	in : INT;
	out : REFERENCE TO UINT;
END_VAR

IF in < DatatypeLimits.MIN_VALUE_OF_INT_WHICH_CAN_BE_HELD_IN_A_UINT THEN
	RETURN;
END_IF

out := INT_TO_UINT(in);
TryConvert_INT_TO_UINT := TRUE;

END_FUNCTION

// mobject-converters/Converters/INT_TO_/TryConvert_INT_TO_UDINT
FUNCTION TryConvert_INT_TO_UDINT : BOOL
VAR_INPUT
	in : INT;
	out : REFERENCE TO UDINT;
END_VAR

IF in < DatatypeLimits.MIN_VALUE_OF_INT_WHICH_CAN_BE_HELD_IN_A_UDINT THEN
	RETURN;
END_IF

out := INT_TO_UDINT(in);
TryConvert_INT_TO_UDINT := TRUE;

END_FUNCTION

// mobject-converters/Converters/INT_TO_/TryConvert_INT_TO_ULINT
FUNCTION TryConvert_INT_TO_ULINT : BOOL
VAR_INPUT
	in : INT;
	out : REFERENCE TO ULINT;
END_VAR

IF in < DatatypeLimits.MIN_VALUE_OF_INT_WHICH_CAN_BE_HELD_IN_A_ULINT THEN
	RETURN;
END_IF

out := INT_TO_ULINT(in);
TryConvert_INT_TO_ULINT := TRUE;

END_FUNCTION

// mobject-converters/Converters/INT_TO_/TryConvert_INT_TO_REAL
FUNCTION TryConvert_INT_TO_REAL : BOOL
VAR_INPUT
	in : INT;
	out : REFERENCE TO REAL;
END_VAR

out := INT_TO_REAL(in);
TryConvert_INT_TO_REAL := TRUE;

END_FUNCTION

// mobject-converters/Converters/INT_TO_/TryConvert_INT_TO_LREAL
FUNCTION TryConvert_INT_TO_LREAL : BOOL
VAR_INPUT
	in : INT;
	out : REFERENCE TO LREAL;
END_VAR

out := INT_TO_LREAL(in);
TryConvert_INT_TO_LREAL := TRUE;

END_FUNCTION

// mobject-converters/Converters/INT_TO_/TryConvert_INT_TO_TIME
FUNCTION TryConvert_INT_TO_TIME : BOOL
VAR_INPUT
	in : INT;
	out : REFERENCE TO TIME;
END_VAR

IF in < DatatypeLimits.MIN_VALUE_OF_INT_WHICH_CAN_BE_HELD_IN_A_TIME THEN
	RETURN;
END_IF

out := INT_TO_TIME(in);
TryConvert_INT_TO_TIME := TRUE;

END_FUNCTION

// mobject-converters/Converters/INT_TO_/TryConvert_INT_TO_TOD
FUNCTION TryConvert_INT_TO_TOD : BOOL
VAR_INPUT
	in : INT;
	out : REFERENCE TO TOD;
END_VAR

IF in < DatatypeLimits.MIN_VALUE_OF_INT_WHICH_CAN_BE_HELD_IN_A_TOD THEN
	RETURN;
END_IF

out := INT_TO_TOD(in);
TryConvert_INT_TO_TOD := TRUE;

END_FUNCTION

// mobject-converters/Converters/INT_TO_/TryConvert_INT_TO_DT
FUNCTION TryConvert_INT_TO_DT : BOOL
VAR_INPUT
	in : INT;
	out : REFERENCE TO DT;
END_VAR

IF in < DatatypeLimits.MIN_VALUE_OF_INT_WHICH_CAN_BE_HELD_IN_A_DT THEN
	RETURN;
END_IF

out := INT_TO_DT(in);
TryConvert_INT_TO_DT := TRUE;

END_FUNCTION

// mobject-converters/Converters/INT_TO_/TryConvert_INT_TO_STRING
FUNCTION TryConvert_INT_TO_STRING : BOOL
VAR_INPUT
	in : INT;
	out : REFERENCE TO STRING;
END_VAR

out := INT_TO_STRING(in);
TryConvert_INT_TO_STRING := TRUE;

END_FUNCTION

// mobject-converters/Converters/LINT_TO_/TryConvert_LINT_TO_BOOL
FUNCTION TryConvert_LINT_TO_BOOL : BOOL
VAR_INPUT
	in : LINT;
	out : REFERENCE TO BOOL;
END_VAR

out := LINT_TO_BOOL(in);
TryConvert_LINT_TO_BOOL := TRUE;

END_FUNCTION

// mobject-converters/Converters/LINT_TO_/TryConvert_LINT_TO_BYTE
FUNCTION TryConvert_LINT_TO_BYTE : BOOL
VAR_INPUT
	in : LINT;
	out : REFERENCE TO BYTE;
END_VAR

IF in > DatatypeLimits.MAX_VALUE_OF_LINT_WHICH_CAN_BE_HELD_IN_A_BYTE THEN
	RETURN;
END_IF

IF in < DatatypeLimits.MIN_VALUE_OF_LINT_WHICH_CAN_BE_HELD_IN_A_BYTE THEN
	RETURN;
END_IF

out := LINT_TO_BYTE(in);
TryConvert_LINT_TO_BYTE := TRUE;

END_FUNCTION

// mobject-converters/Converters/LINT_TO_/TryConvert_LINT_TO_DATE
FUNCTION TryConvert_LINT_TO_DATE : BOOL
VAR_INPUT
	in : LINT;
	out : REFERENCE TO DATE;
END_VAR

IF in > DatatypeLimits.MAX_VALUE_OF_LINT_WHICH_CAN_BE_HELD_IN_A_DATE THEN
	RETURN;
END_IF

IF in < DatatypeLimits.MIN_VALUE_OF_LINT_WHICH_CAN_BE_HELD_IN_A_DATE THEN
	RETURN;
END_IF

out := LINT_TO_DATE(in);
TryConvert_LINT_TO_DATE := TRUE;

END_FUNCTION

// mobject-converters/Converters/LINT_TO_/TryConvert_LINT_TO_Destination
FUNCTION TryConvert_LINT_TO_Destination : BOOL
VAR_INPUT
	in : LINT;
	out : ANY;
END_VAR
VAR
	convertResult : BOOL := FALSE;
	convertAddress : PVOID;
	_BOOL : BOOL;
	_BYTE : BYTE;
	_WORD : WORD;
	_DWORD : DWORD;
	_LWORD : LWORD;
	_SINT : SINT;
	_INT : INT;
	_DINT : DINT;
	_LINT : LINT;
	_USINT : USINT;
	_UINT : UINT;
	_UDINT : UDINT;
	_ULINT : ULINT;
	_REAL : REAL;
	_LREAL : LREAL;
	_TIME : TIME;
	_TOD : TOD;
	_DATE : DATE;
	_DT : DT;
	_STRING : STRING;
END_VAR

CASE out.TypeClass OF
	__SYSTEM.TYPE_CLASS.TYPE_BOOL:
	
	convertResult := TryConvert_LINT_TO_BOOL(in, _BOOL);
	IF convertResult THEN
		convertAddress := ADR(_BOOL);
	END_IF
	
	__SYSTEM.TYPE_CLASS.TYPE_BYTE:
	
	convertResult := TryConvert_LINT_TO_BYTE(in, _BYTE);
	IF convertResult THEN
		convertAddress := ADR(_BYTE);
	END_IF
	
	__SYSTEM.TYPE_CLASS.TYPE_WORD:
	
	convertResult := TryConvert_LINT_TO_WORD(in, _WORD);
	IF convertResult THEN
		convertAddress := ADR(_WORD);
	END_IF
	
	__SYSTEM.TYPE_CLASS.TYPE_DWORD:
	
	convertResult := TryConvert_LINT_TO_DWORD(in, _DWORD);
	IF convertResult THEN
		convertAddress := ADR(_DWORD);
	END_IF
	
	__SYSTEM.TYPE_CLASS.TYPE_LWORD:
	
	convertResult := TryConvert_LINT_TO_LWORD(in, _LWORD);
	IF convertResult THEN
		convertAddress := ADR(_LWORD);
	END_IF
	
	__SYSTEM.TYPE_CLASS.TYPE_SINT:
	
	convertResult := TryConvert_LINT_TO_SINT(in, _SINT);
	IF convertResult THEN
		convertAddress := ADR(_SINT);
	END_IF
	
	__SYSTEM.TYPE_CLASS.TYPE_INT:
	
	convertResult := TryConvert_LINT_TO_INT(in, _INT);
	IF convertResult THEN
		convertAddress := ADR(_INT);
	END_IF
	
	__SYSTEM.TYPE_CLASS.TYPE_DINT:
	
	convertResult := TryConvert_LINT_TO_DINT(in, _DINT);
	IF convertResult THEN
		convertAddress := ADR(_DINT);
	END_IF
	
	__SYSTEM.TYPE_CLASS.TYPE_LINT:
	
	convertResult := TryConvert_LINT_TO_LINT(in, _LINT);
	IF convertResult THEN
		convertAddress := ADR(_LINT);
	END_IF
	
	__SYSTEM.TYPE_CLASS.TYPE_USINT:
	
	convertResult := TryConvert_LINT_TO_USINT(in, _USINT);
	IF convertResult THEN
		convertAddress := ADR(_USINT);
	END_IF
	
	__SYSTEM.TYPE_CLASS.TYPE_UINT:
	
	convertResult := TryConvert_LINT_TO_UINT(in, _UINT);
	IF convertResult THEN
		convertAddress := ADR(_UINT);
	END_IF
	
	__SYSTEM.TYPE_CLASS.TYPE_UDINT:
	
	convertResult := TryConvert_LINT_TO_UDINT(in, _UDINT);
	IF convertResult THEN
		convertAddress := ADR(_UDINT);
	END_IF
	
	__SYSTEM.TYPE_CLASS.TYPE_ULINT:
	
	convertResult := TryConvert_LINT_TO_ULINT(in, _ULINT);
	IF convertResult THEN
		convertAddress := ADR(_ULINT);
	END_IF
	
	__SYSTEM.TYPE_CLASS.TYPE_REAL:
	
	convertResult := TryConvert_LINT_TO_REAL(in, _REAL);
	IF convertResult THEN
		convertAddress := ADR(_REAL);
	END_IF
	
	__SYSTEM.TYPE_CLASS.TYPE_LREAL:
	
	convertResult := TryConvert_LINT_TO_LREAL(in, _LREAL);
	IF convertResult THEN
		convertAddress := ADR(_LREAL);
	END_IF
	
	__SYSTEM.TYPE_CLASS.TYPE_TIME:
	
	convertResult := TryConvert_LINT_TO_TIME(in, _TIME);
	IF convertResult THEN
		convertAddress := ADR(_TIME);
	END_IF
	
	__SYSTEM.TYPE_CLASS.TYPE_TIMEOFDAY:
	
	convertResult := TryConvert_LINT_TO_TOD(in, _TOD);
	IF convertResult THEN
		convertAddress := ADR(_TOD);
	END_IF
	
	__SYSTEM.TYPE_CLASS.TYPE_DATE:
	
	convertResult := TryConvert_LINT_TO_DATE(in, _DATE);
	IF convertResult THEN
		convertAddress := ADR(_DATE);
	END_IF
	
	__SYSTEM.TYPE_CLASS.TYPE_DATEANDTIME:
	
	convertResult := TryConvert_LINT_TO_DT(in, _DT);
	IF convertResult THEN
		convertAddress := ADR(_DT);
	END_IF
	
